RoboDK station: kr30 cnc template half inch flat end mill - paulina 2.rdk

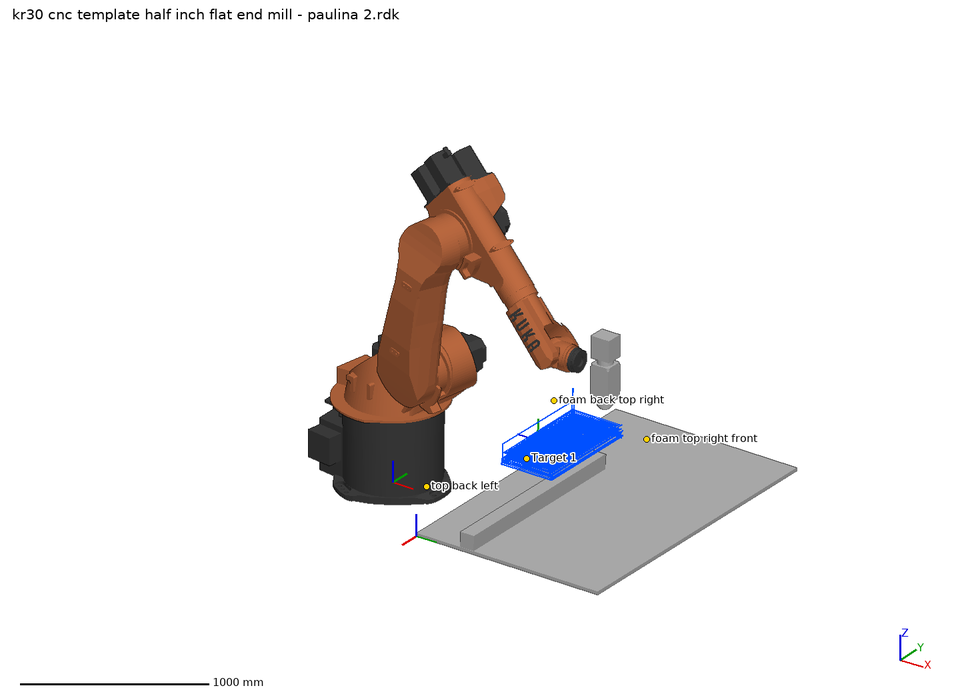
[picture v0: the station drawn from its stored meshes, robots at their saved joint values, targets as dots, program paths as lines]
Station kr30 cnc template half inch flat end mill - paulina 2. Poses are relative to the parent item; angles as X-Y-Z fixed-axis rotations.
  - frame KUKA KR 30 HA Base at (0, 0, 0) mm
    - robot KUKA KR 30 HA: 6 axes, payload 30 kg, reach 2033 mm, repeatability 0.05 mm, weight 665 kg
        modified DH rows (alpha deg, a mm, theta deg, d mm): 0, 0, 0, 815; -90, 350, 0, 0; 0, 850, -90, 0; -90, 145, 0, 820; 90, 0, 0, 0; -90, 0, 180, 170
        joint limits [-185, -135, -120, -350, -119, -350] to [185, 35, 158, 350, 119, 350]; home [0, -90, 90, 0, 0, 0]; saved at [10.988, -78.154, 121.402, 16.012, -43.574, -11.346]
      - tool rc90 spindle mm, TCP at (337.31, -2.2, 160.57) mm, size 110 x 421.3 x 118 mm, geometry from rc90 spindle mm.stl
    - frame Tabletop at (921.82, -1104.91, 385) mm, rotated rx -0.93 ry -0.21 rz -89.9 deg
      - object tabletop CHECK HEIGHT at (-1839.9, 0, 0) mm, size 1839.9 x 1168.4 x 19 mm, geometry from kr30 tabletop mm.stl
      - object kr30 pipe jig base at (-1220, -610.6, 0) mm, size 1217.6 x 88.9 x 88.9 mm, geometry from kr30 pipe jig base.stl
      - frame Frame 3 at (-550, 390, 460) mm, rotated rx 90 ry 0 rz 0 deg
        - target Target 1 (Cartesian target) at (324.46, 69.12, -153.95) mm, rotated rx -179.9 ry 0.14 rz -89.96 deg; joints [37.245, -66.694, 101.534, 53.768, -48.608, -41.204] of KUKA KR 30 HA
    - target foam back top right (Cartesian target) at (1197.65, -230.62, 906.79) mm, rotated rx -15.53 ry 90 rz -15.53 deg; joints [14.757, -102.447, 141.256, 22.791, -41.102, -17.568] of KUKA KR 30 HA
    - target foam top right front (Cartesian target) at (1797.45, -230.62, 850.68) mm, rotated rx -15.58 ry 90 rz -15.58 deg; joints [8.85, -62.405, 99.608, 14.434, -38.093, -11.451] of KUKA KR 30 HA
    - target top back left (Cartesian target) at (1223.08, -1440.01, 894.96) mm, rotated rx 58.97 ry 90 rz 58.97 deg; joints [58.171, -50.232, 76.73, 74.515, -61.834, -59.599] of KUKA KR 30 HA
  - machining project Machining Settings: C:/Users/Research Office/Downloads/B.apt | rotZ(0) | rotX(0)*rotY(0) | roty(-90)
  - program Machining (5196 instructions, listed below)
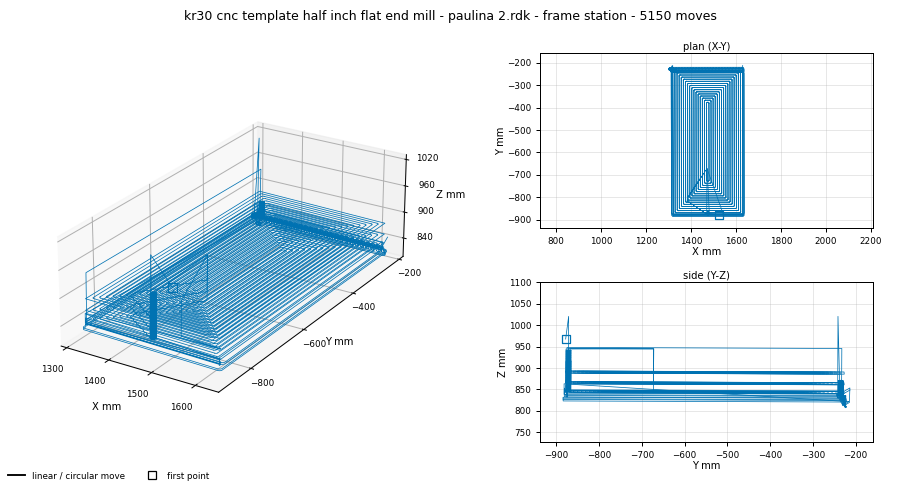
[picture p0: tool path of kr30 cnc template half inch flat end mill - paulina 2.rdk in frame station, 5150 of 5150 moves have a stored position in this frame; points joined in program order, loops and branches not executed]

--- program Machining (robot KUKA KR 30 HA) ---
  Smooth(15)
  Print: /'1001'
  Print: /''
  Print: /'Pocket1'
  Call SetTool(1)
  Set speed (1000.0 mm/s)
  Set Ref.: Frame 3
  Set Tool: rc90 spindle mm
  Show rc90 spindle mm
  MoveJ 1 to (326.02, 133.41, -204.56) mm, rotated rx -179.9 ry 0.15 rz -89.95 deg; joints [36.075, -65.683, 95.357, 56.596, -44.843, -46.24]
  MoveL 2 to (319.15, 185.52, -150.09) mm, rotated rx -179.9 ry 0 rz -90 deg; joints [37.098, -69.807, 97.257, -120.358, 44.337, 130.231]
  MoveL 3 to (319.15, 185.52, -150.09) mm, rotated rx -179.9 ry 0 rz -90 deg; joints [37.098, -69.807, 97.257, -120.358, 44.337, 130.231]
  Set speed (1000.0 mm/s)
  MoveL 4 to (319.15, 108.04, -150.09) mm, rotated rx -179.9 ry 0 rz -90 deg; joints [37.137, -68.08, 100.527, -124.443, 47.047, 136.103]
  Set speed (100.0 mm/s)
  MoveL 5 to (319.13, 107.83, -150.09) mm, rotated rx -179.9 ry 0 rz -90 deg; joints [37.137, -68.075, 100.537, -124.454, 47.054, 136.119]
  MoveL 6 to (319.08, 107.62, -150.09) mm, rotated rx -179.9 ry 0 rz -90 deg; joints [37.135, -68.072, 100.548, -124.467, 47.061, 136.136]
  MoveL 7 to (318.99, 107.42, -150.09) mm, rotated rx -179.9 ry 0 rz -90 deg; joints [37.132, -68.071, 100.56, -124.48, 47.067, 136.154]
  MoveL 8 to (318.86, 107.24, -150.09) mm, rotated rx -179.9 ry 0 rz -90 deg; joints [37.129, -68.071, 100.574, -124.494, 47.072, 136.171]
  MoveL 9 to (318.71, 107.09, -150.1) mm, rotated rx -179.9 ry 0 rz -90 deg; joints [37.124, -68.072, 100.587, -124.508, 47.076, 136.188]
  MoveL 10 to (318.54, 106.96, -150.11) mm, rotated rx -179.9 ry 0 rz -90 deg; joints [37.118, -68.075, 100.601, -124.522, 47.078, 136.204]
  MoveL 11 to (318.35, 106.86, -150.13) mm, rotated rx -179.9 ry 0 rz -90 deg; joints [37.111, -68.078, 100.613, -124.535, 47.078, 136.218]
  MoveL 12 to (318.14, 106.8, -150.16) mm, rotated rx -179.9 ry 0 rz -90 deg; joints [37.104, -68.083, 100.625, -124.547, 47.077, 136.23]
  MoveL 13 to (317.93, 106.77, -150.19) mm, rotated rx -179.9 ry 0 rz -90 deg; joints [37.097, -68.089, 100.634, -124.558, 47.074, 136.24]
  MoveL 14 to (315.89, 106.7, -150.99) mm, rotated rx -179.9 ry 0 rz -90 deg; joints [37.013, -68.123, 100.691, -124.657, 47.028, 136.319]
  MoveL 15 to (314.27, 106.62, -152.45) mm, rotated rx -179.9 ry 0 rz -90 deg; joints [36.926, -68.109, 100.678, -124.744, 46.969, 136.378]
  MoveL 16 to (313.28, 106.54, -154.4) mm, rotated rx -179.9 ry 0 rz -90 deg; joints [36.848, -68.046, 100.598, -124.808, 46.905, 136.41]
  MoveL 17 to (313.05, 106.47, -156.57) mm, rotated rx -179.9 ry 0 rz -90 deg; joints [36.788, -67.944, 100.461, -124.84, 46.845, 136.411]
  MoveL 18 to (313.61, 106.39, -158.69) mm, rotated rx -179.9 ry 0 rz -90 deg; joints [36.756, -67.815, 100.287, -124.838, 46.796, 136.381]
  MoveL 19 to (314.88, 106.31, -160.46) mm, rotated rx -179.9 ry 0 rz -90 deg; joints [36.754, -67.676, 100.098, -124.8, 46.766, 136.325]
  MoveL 20 to (316.71, 106.24, -161.67) mm, rotated rx -179.9 ry 0 rz -90 deg; joints [36.783, -67.546, 99.919, -124.734, 46.759, 136.252]
  MoveL 21 to (318.84, 106.16, -162.15) mm, rotated rx -179.9 ry 0 rz -90 deg; joints [36.84, -67.44, 99.775, -124.649, 46.776, 136.171]
  MoveL 22 to (321, 106.08, -161.83) mm, rotated rx -179.9 ry 0 rz -90 deg; joints [36.915, -67.373, 99.684, -124.556, 46.815, 136.094]
  MoveL 23 to (322.91, 106.01, -160.77) mm, rotated rx -179.9 ry 0 rz -90 deg; joints [37.001, -67.353, 99.659, -124.468, 46.872, 136.033]
  MoveL 24 to (324.31, 105.93, -159.1) mm, rotated rx -179.9 ry 0 rz -90 deg; joints [37.085, -67.382, 99.704, -124.397, 46.94, 135.995]
  MoveL 25 to (325.03, 105.85, -157.03) mm, rotated rx -179.9 ry 0 rz -90 deg; joints [37.158, -67.457, 99.813, -124.353, 47.009, 135.987]
  MoveL 26 to (324.97, 105.78, -154.85) mm, rotated rx -179.9 ry 0 rz -90 deg; joints [37.208, -67.566, 99.972, -124.342, 47.072, 136.01]
  MoveL 27 to (324.13, 105.7, -152.83) mm, rotated rx -179.9 ry 0 rz -90 deg; joints [37.23, -67.697, 100.161, -124.365, 47.121, 136.061]
  MoveL 28 to (322.62, 105.62, -151.24) mm, rotated rx -179.9 ry 0 rz -90 deg; joints [37.221, -67.831, 100.355, -124.42, 47.148, 136.135]
  MoveL 29 to (320.65, 105.55, -150.3) mm, rotated rx -179.9 ry 0 rz -90 deg; joints [37.181, -67.95, 100.529, -124.501, 47.152, 136.222]
  MoveL 30 to (318.48, 105.47, -150.11) mm, rotated rx -179.9 ry 0 rz -90 deg; joints [37.117, -68.039, 100.661, -124.597, 47.131, 136.313]
  MoveL 31 to (316.38, 105.39, -150.72) mm, rotated rx -179.9 ry 0 rz -90 deg; joints [37.035, -68.086, 100.734, -124.697, 47.09, 136.396]
  MoveL 32 to (314.63, 105.32, -152.03) mm, rotated rx -179.9 ry 0 rz -90 deg; joints [36.948, -68.084, 100.739, -124.788, 47.034, 136.46]
  MoveL 33 to (313.47, 105.24, -153.88) mm, rotated rx -179.9 ry 0 rz -90 deg; joints [36.867, -68.033, 100.675, -124.859, 46.97, 136.499]
  MoveL 34 to (313.04, 105.16, -156.02) mm, rotated rx -179.9 ry 0 rz -90 deg; joints [36.802, -67.939, 100.551, -124.9, 46.908, 136.508]
  MoveL 35 to (313.4, 105.09, -158.18) mm, rotated rx -179.9 ry 0 rz -90 deg; joints [36.762, -67.816, 100.385, -124.906, 46.856, 136.486]
  MoveL 36 to (314.5, 105.01, -160.06) mm, rotated rx -179.9 ry 0 rz -90 deg; joints [36.752, -67.678, 100.197, -124.877, 46.82, 136.436]
  MoveL 37 to (316.21, 104.93, -161.43) mm, rotated rx -179.9 ry 0 rz -90 deg; joints [36.774, -67.544, 100.013, -124.818, 46.807, 136.366]
  MoveL 38 to (318.29, 104.86, -162.1) mm, rotated rx -179.9 ry 0 rz -90 deg; joints [36.824, -67.43, 99.858, -124.736, 46.818, 136.286]
  MoveL 39 to (320.47, 104.78, -161.99) mm, rotated rx -179.9 ry 0 rz -90 deg; joints [36.896, -67.353, 99.752, -124.644, 46.852, 136.207]
  MoveL 40 to (322.47, 104.7, -161.1) mm, rotated rx -179.9 ry 0 rz -90 deg; joints [36.98, -67.32, 99.71, -124.553, 46.905, 136.141]
  MoveL 41 to (324.02, 104.63, -159.56) mm, rotated rx -179.9 ry 0 rz -90 deg; joints [37.066, -67.337, 99.738, -124.477, 46.97, 136.097]
  MoveL 42 to (324.92, 104.55, -157.57) mm, rotated rx -179.9 ry 0 rz -90 deg; joints [37.142, -67.401, 99.832, -124.426, 47.04, 136.081]
  MoveL 43 to (325.06, 104.47, -155.39) mm, rotated rx -179.9 ry 0 rz -90 deg; joints [37.198, -67.503, 99.98, -124.406, 47.106, 136.096]
  MoveL 44 to (324.41, 104.4, -153.31) mm, rotated rx -179.9 ry 0 rz -90 deg; joints [37.228, -67.63, 100.163, -124.42, 47.159, 136.141]
  MoveL 45 to (323.06, 104.32, -151.59) mm, rotated rx -179.9 ry 0 rz -90 deg; joints [37.227, -67.764, 100.359, -124.467, 47.192, 136.21]
  MoveL 46 to (321.18, 104.24, -150.47) mm, rotated rx -179.9 ry 0 rz -90 deg; joints [37.195, -67.889, 100.54, -124.542, 47.202, 136.295]
  MoveL 47 to (319.03, 104.17, -150.09) mm, rotated rx -179.9 ry 0 rz -90 deg; joints [37.136, -67.987, 100.685, -124.636, 47.187, 136.385]
  MoveL 48 to (316.88, 104.09, -150.49) mm, rotated rx -179.9 ry 0 rz -90 deg; joints [37.058, -68.045, 100.774, -124.736, 47.151, 136.471]
  MoveL 49 to (315.02, 104.01, -151.64) mm, rotated rx -179.9 ry 0 rz -90 deg; joints [36.971, -68.055, 100.796, -124.831, 47.098, 136.541]
  MoveL 50 to (313.7, 103.94, -153.37) mm, rotated rx -179.9 ry 0 rz -90 deg; joints [36.887, -68.016, 100.749, -124.908, 47.035, 136.587]
  MoveL 51 to (313.07, 103.86, -155.47) mm, rotated rx -179.9 ry 0 rz -90 deg; joints [36.817, -67.933, 100.639, -124.957, 46.972, 136.604]
  MoveL 52 to (313.23, 103.78, -157.65) mm, rotated rx -179.9 ry 0 rz -90 deg; joints [36.77, -67.815, 100.481, -124.972, 46.916, 136.589]
  MoveL 53 to (314.16, 103.71, -159.63) mm, rotated rx -179.9 ry 0 rz -90 deg; joints [36.752, -67.68, 100.296, -124.952, 46.876, 136.546]
  MoveL 54 to (315.73, 103.63, -161.14) mm, rotated rx -179.9 ry 0 rz -90 deg; joints [36.766, -67.543, 100.109, -124.9, 46.857, 136.48]
  MoveL 55 to (317.74, 103.55, -162) mm, rotated rx -179.9 ry 0 rz -90 deg; joints [36.809, -67.423, 99.945, -124.823, 46.861, 136.401]
  MoveL 56 to (319.92, 103.48, -162.09) mm, rotated rx -179.9 ry 0 rz -90 deg; joints [36.877, -67.335, 99.825, -124.732, 46.889, 136.321]
  MoveL 57 to (322, 103.4, -161.39) mm, rotated rx -179.9 ry 0 rz -90 deg; joints [36.959, -67.291, 99.766, -124.639, 46.938, 136.251]
  MoveL 58 to (323.68, 103.32, -160) mm, rotated rx -179.9 ry 0 rz -90 deg; joints [37.045, -67.295, 99.775, -124.559, 47.001, 136.2]
  MoveL 59 to (324.76, 103.25, -158.11) mm, rotated rx -179.9 ry 0 rz -90 deg; joints [37.125, -67.348, 99.853, -124.5, 47.071, 136.177]
  MoveL 60 to (325.1, 103.17, -155.95) mm, rotated rx -179.9 ry 0 rz -90 deg; joints [37.187, -67.441, 99.989, -124.471, 47.138, 136.184]
  MoveL 61 to (324.64, 103.09, -153.81) mm, rotated rx -179.9 ry 0 rz -90 deg; joints [37.224, -67.563, 100.166, -124.477, 47.195, 136.222]
  MoveL 62 to (323.45, 103.02, -151.98) mm, rotated rx -179.9 ry 0 rz -90 deg; joints [37.231, -67.697, 100.361, -124.517, 47.234, 136.285]
  MoveL 63 to (321.69, 102.94, -150.69) mm, rotated rx -179.9 ry 0 rz -90 deg; joints [37.206, -67.826, 100.548, -124.585, 47.25, 136.367]
  MoveL 64 to (319.58, 102.86, -150.11) mm, rotated rx -179.9 ry 0 rz -90 deg; joints [37.153, -67.932, 100.704, -124.675, 47.242, 136.457]
  MoveL 65 to (317.41, 102.79, -150.32) mm, rotated rx -179.9 ry 0 rz -90 deg; joints [37.079, -68.001, 100.808, -124.775, 47.211, 136.545]
  MoveL 66 to (315.45, 102.71, -151.29) mm, rotated rx -179.9 ry 0 rz -90 deg; joints [36.994, -68.024, 100.848, -124.872, 47.161, 136.62]
  MoveL 67 to (313.97, 102.63, -152.89) mm, rotated rx -179.9 ry 0 rz -90 deg; joints [36.908, -67.997, 100.818, -124.955, 47.1, 136.673]
  MoveL 68 to (313.16, 102.56, -154.92) mm, rotated rx -179.9 ry 0 rz -90 deg; joints [36.833, -67.924, 100.723, -125.012, 47.037, 136.697]
  MoveL 69 to (313.12, 102.48, -157.11) mm, rotated rx -179.9 ry 0 rz -90 deg; joints [36.78, -67.814, 100.575, -125.036, 46.978, 136.69]
  MoveL 70 to (313.86, 102.4, -159.16) mm, rotated rx -179.9 ry 0 rz -90 deg; joints [36.754, -67.681, 100.395, -125.025, 46.933, 136.654]
  MoveL 71 to (315.29, 102.33, -160.82) mm, rotated rx -179.9 ry 0 rz -90 deg; joints [36.76, -67.543, 100.206, -124.98, 46.908, 136.593]
  MoveL 72 to (317.21, 102.25, -161.86) mm, rotated rx -179.9 ry 0 rz -90 deg; joints [36.797, -67.417, 100.034, -124.908, 46.907, 136.516]
  MoveL 73 to (319.37, 102.17, -162.14) mm, rotated rx -179.9 ry 0 rz -90 deg; joints [36.859, -67.32, 99.901, -124.819, 46.929, 136.435]
  MoveL 74 to (321.5, 102.1, -161.64) mm, rotated rx -179.9 ry 0 rz -90 deg; joints [36.938, -67.264, 99.825, -124.726, 46.973, 136.361]
  MoveL 75 to (323.31, 102.02, -160.41) mm, rotated rx -179.9 ry 0 rz -90 deg; joints [37.024, -67.256, 99.818, -124.641, 47.033, 136.305]
  MoveL 76 to (324.56, 101.94, -158.62) mm, rotated rx -179.9 ry 0 rz -90 deg; joints [37.107, -67.297, 99.879, -124.576, 47.102, 136.274]
  MoveL 77 to (325.09, 101.86, -156.5) mm, rotated rx -179.9 ry 0 rz -90 deg; joints [37.174, -67.381, 100.002, -124.539, 47.17, 136.274]
  MoveL 78 to (324.83, 101.79, -154.33) mm, rotated rx -179.9 ry 0 rz -90 deg; joints [37.218, -67.497, 100.17, -124.536, 47.231, 136.304]
  MoveL 79 to (323.82, 101.71, -152.4) mm, rotated rx -179.9 ry 0 rz -90 deg; joints [37.233, -67.63, 100.363, -124.567, 47.275, 136.361]
  MoveL 80 to (322.18, 101.63, -150.95) mm, rotated rx -179.9 ry 0 rz -90 deg; joints [37.216, -67.761, 100.554, -124.629, 47.297, 136.439]
  MoveL 81 to (320.13, 101.56, -150.18) mm, rotated rx -179.9 ry 0 rz -90 deg; joints [37.17, -67.875, 100.72, -124.715, 47.295, 136.528]
  MoveL 82 to (317.95, 101.48, -150.19) mm, rotated rx -179.9 ry 0 rz -90 deg; joints [37.1, -67.954, 100.839, -124.813, 47.269, 136.618]
  MoveL 83 to (315.91, 101.4, -150.98) mm, rotated rx -179.9 ry 0 rz -90 deg; joints [37.016, -67.989, 100.896, -124.912, 47.224, 136.697]
  MoveL 84 to (314.29, 101.33, -152.44) mm, rotated rx -179.9 ry 0 rz -90 deg; joints [36.929, -67.975, 100.883, -125, 47.166, 136.756]
  MoveL 85 to (313.29, 101.25, -154.38) mm, rotated rx -179.9 ry 0 rz -90 deg; joints [36.851, -67.913, 100.804, -125.064, 47.102, 136.788]
  MoveL 86 to (313.05, 101.17, -156.56) mm, rotated rx -179.9 ry 0 rz -90 deg; joints [36.792, -67.811, 100.668, -125.097, 47.041, 136.789]
  MoveL 87 to (313.6, 101.1, -158.67) mm, rotated rx -179.9 ry 0 rz -90 deg; joints [36.759, -67.682, 100.493, -125.095, 46.992, 136.76]
  MoveL 88 to (314.87, 101.02, -160.45) mm, rotated rx -179.9 ry 0 rz -90 deg; joints [36.757, -67.544, 100.304, -125.058, 46.962, 136.704]
  MoveL 89 to (316.69, 100.94, -161.66) mm, rotated rx -179.9 ry 0 rz -90 deg; joints [36.786, -67.414, 100.125, -124.992, 46.954, 136.631]
  MoveL 90 to (318.82, 100.87, -162.14) mm, rotated rx -179.9 ry 0 rz -90 deg; joints [36.842, -67.308, 99.981, -124.907, 46.97, 136.55]
  MoveL 91 to (320.98, 100.79, -161.84) mm, rotated rx -179.9 ry 0 rz -90 deg; joints [36.917, -67.241, 99.889, -124.813, 47.008, 136.473]
  MoveL 92 to (322.89, 100.71, -160.78) mm, rotated rx -179.9 ry 0 rz -90 deg; joints [37.003, -67.22, 99.864, -124.725, 47.065, 136.411]
  MoveL 93 to (324.3, 100.64, -159.11) mm, rotated rx -179.9 ry 0 rz -90 deg; joints [37.087, -67.249, 99.908, -124.654, 47.132, 136.374]
  MoveL 94 to (325.03, 100.56, -157.05) mm, rotated rx -179.9 ry 0 rz -90 deg; joints [37.16, -67.323, 100.017, -124.609, 47.202, 136.365]
  MoveL 95 to (324.97, 100.48, -154.87) mm, rotated rx -179.9 ry 0 rz -90 deg; joints [37.21, -67.432, 100.175, -124.597, 47.265, 136.388]
  MoveL 96 to (324.14, 100.41, -152.85) mm, rotated rx -179.9 ry 0 rz -90 deg; joints [37.233, -67.562, 100.364, -124.62, 47.314, 136.439]
  MoveL 97 to (322.64, 100.33, -151.26) mm, rotated rx -179.9 ry 0 rz -90 deg; joints [37.224, -67.696, 100.558, -124.675, 47.342, 136.513]
  MoveL 98 to (320.67, 100.25, -150.3) mm, rotated rx -179.9 ry 0 rz -90 deg; joints [37.184, -67.815, 100.733, -124.755, 47.346, 136.6]
  MoveL 99 to (318.5, 100.18, -150.11) mm, rotated rx -179.9 ry 0 rz -90 deg; joints [37.12, -67.904, 100.865, -124.851, 47.327, 136.69]
  MoveL 100 to (316.39, 100.1, -150.71) mm, rotated rx -179.9 ry 0 rz -90 deg; joints [37.039, -67.951, 100.939, -124.952, 47.286, 136.773]
  MoveL 101 to (314.64, 100.02, -152.02) mm, rotated rx -179.9 ry 0 rz -90 deg; joints [36.952, -67.949, 100.944, -125.043, 47.23, 136.838]
  MoveL 102 to (313.47, 99.95, -153.86) mm, rotated rx -179.9 ry 0 rz -90 deg; joints [36.87, -67.899, 100.88, -125.114, 47.167, 136.877]
  MoveL 103 to (313.04, 99.87, -156) mm, rotated rx -179.9 ry 0 rz -90 deg; joints [36.805, -67.806, 100.757, -125.156, 47.105, 136.886]
  MoveL 104 to (313.39, 99.79, -158.16) mm, rotated rx -179.9 ry 0 rz -90 deg; joints [36.765, -67.683, 100.591, -125.163, 47.052, 136.864]
  MoveL 105 to (314.49, 99.72, -160.05) mm, rotated rx -179.9 ry 0 rz -90 deg; joints [36.755, -67.545, 100.403, -125.134, 47.016, 136.815]
  MoveL 106 to (316.19, 99.64, -161.42) mm, rotated rx -179.9 ry 0 rz -90 deg; joints [36.776, -67.411, 100.219, -125.075, 47.002, 136.745]
  MoveL 107 to (318.27, 99.56, -162.1) mm, rotated rx -179.9 ry 0 rz -90 deg; joints [36.826, -67.298, 100.064, -124.993, 47.012, 136.664]
  MoveL 108 to (320.45, 99.49, -161.99) mm, rotated rx -179.9 ry 0 rz -90 deg; joints [36.898, -67.22, 99.957, -124.901, 47.045, 136.585]
  MoveL 109 to (322.45, 99.41, -161.11) mm, rotated rx -179.9 ry 0 rz -90 deg; joints [36.982, -67.187, 99.915, -124.81, 47.098, 136.519]
  MoveL 110 to (324.01, 99.33, -159.58) mm, rotated rx -179.9 ry 0 rz -90 deg; joints [37.068, -67.204, 99.941, -124.733, 47.163, 136.475]
  MoveL 111 to (324.92, 99.26, -157.59) mm, rotated rx -179.9 ry 0 rz -90 deg; joints [37.144, -67.267, 100.035, -124.681, 47.233, 136.459]
  MoveL 112 to (325.06, 99.18, -155.41) mm, rotated rx -179.9 ry 0 rz -90 deg; joints [37.201, -67.368, 100.182, -124.661, 47.299, 136.474]
  MoveL 113 to (324.42, 99.1, -153.33) mm, rotated rx -179.9 ry 0 rz -90 deg; joints [37.231, -67.494, 100.366, -124.675, 47.352, 136.518]
  MoveL 114 to (323.07, 99.03, -151.6) mm, rotated rx -179.9 ry 0 rz -90 deg; joints [37.23, -67.629, 100.561, -124.722, 47.386, 136.586]
  MoveL 115 to (321.2, 98.95, -150.47) mm, rotated rx -179.9 ry 0 rz -90 deg; joints [37.198, -67.753, 100.743, -124.796, 47.396, 136.671]
  MoveL 116 to (319.05, 98.87, -150.09) mm, rotated rx -179.9 ry 0 rz -90 deg; joints [37.139, -67.851, 100.888, -124.89, 47.383, 136.762]
  MoveL 117 to (316.9, 98.8, -150.49) mm, rotated rx -179.9 ry 0 rz -90 deg; joints [37.061, -67.91, 100.977, -124.99, 47.347, 136.847]
  MoveL 118 to (315.04, 98.72, -151.63) mm, rotated rx -179.9 ry 0 rz -90 deg; joints [36.974, -67.92, 101, -125.085, 47.295, 136.917]
  MoveL 119 to (313.7, 98.64, -153.36) mm, rotated rx -179.9 ry 0 rz -90 deg; joints [36.89, -67.882, 100.953, -125.162, 47.232, 136.964]
  MoveL 120 to (313.07, 98.57, -155.45) mm, rotated rx -179.9 ry 0 rz -90 deg; joints [36.82, -67.799, 100.844, -125.212, 47.169, 136.981]
  MoveL 121 to (313.23, 98.49, -157.63) mm, rotated rx -179.9 ry 0 rz -90 deg; joints [36.773, -67.682, 100.686, -125.228, 47.113, 136.966]
  MoveL 122 to (314.15, 98.41, -159.61) mm, rotated rx -179.9 ry 0 rz -90 deg; joints [36.755, -67.546, 100.502, -125.208, 47.073, 136.923]
  MoveL 123 to (315.72, 98.34, -161.13) mm, rotated rx -179.9 ry 0 rz -90 deg; joints [36.769, -67.41, 100.314, -125.156, 47.053, 136.858]
  MoveL 124 to (317.72, 98.26, -162) mm, rotated rx -179.9 ry 0 rz -90 deg; joints [36.812, -67.29, 100.15, -125.079, 47.056, 136.779]
  MoveL 125 to (319.91, 98.18, -162.09) mm, rotated rx -179.9 ry 0 rz -90 deg; joints [36.879, -67.202, 100.029, -124.988, 47.084, 136.699]
  MoveL 126 to (321.98, 98.11, -161.4) mm, rotated rx -179.9 ry 0 rz -90 deg; joints [36.961, -67.157, 99.97, -124.896, 47.132, 136.628]
  MoveL 127 to (323.67, 98.03, -160.02) mm, rotated rx -179.9 ry 0 rz -90 deg; joints [37.047, -67.161, 99.979, -124.814, 47.194, 136.577]
  MoveL 128 to (324.76, 97.95, -158.12) mm, rotated rx -179.9 ry 0 rz -90 deg; joints [37.127, -67.213, 100.056, -124.755, 47.264, 136.554]
  MoveL 129 to (325.1, 97.88, -155.97) mm, rotated rx -179.9 ry 0 rz -90 deg; joints [37.189, -67.306, 100.192, -124.726, 47.332, 136.561]
  MoveL 130 to (324.65, 97.8, -153.83) mm, rotated rx -179.9 ry 0 rz -90 deg; joints [37.227, -67.427, 100.368, -124.731, 47.389, 136.598]
  MoveL 131 to (323.47, 97.72, -151.99) mm, rotated rx -179.9 ry 0 rz -90 deg; joints [37.233, -67.561, 100.563, -124.77, 47.428, 136.661]
  MoveL 132 to (321.71, 97.65, -150.69) mm, rotated rx -179.9 ry 0 rz -90 deg; joints [37.209, -67.69, 100.75, -124.838, 47.445, 136.743]
  MoveL 133 to (319.6, 97.57, -150.11) mm, rotated rx -179.9 ry 0 rz -90 deg; joints [37.157, -67.796, 100.906, -124.928, 47.437, 136.833]
  MoveL 134 to (317.43, 97.49, -150.31) mm, rotated rx -179.9 ry 0 rz -90 deg; joints [37.083, -67.865, 101.011, -125.028, 47.407, 136.921]
  MoveL 135 to (315.47, 97.41, -151.28) mm, rotated rx -179.9 ry 0 rz -90 deg; joints [36.997, -67.888, 101.051, -125.125, 47.358, 136.996]
  MoveL 136 to (313.98, 97.34, -152.88) mm, rotated rx -179.9 ry 0 rz -90 deg; joints [36.911, -67.862, 101.022, -125.208, 47.298, 137.049]
  MoveL 137 to (313.16, 97.26, -154.9) mm, rotated rx -179.9 ry 0 rz -90 deg; joints [36.837, -67.789, 100.927, -125.266, 47.234, 137.073]
  MoveL 138 to (313.11, 97.18, -157.09) mm, rotated rx -179.9 ry 0 rz -90 deg; joints [36.783, -67.68, 100.78, -125.291, 47.176, 137.067]
  MoveL 139 to (313.85, 97.11, -159.14) mm, rotated rx -179.9 ry 0 rz -90 deg; joints [36.757, -67.547, 100.6, -125.28, 47.13, 137.03]
  MoveL 140 to (315.27, 97.03, -160.8) mm, rotated rx -179.9 ry 0 rz -90 deg; joints [36.763, -67.409, 100.411, -125.236, 47.105, 136.97]
  MoveL 141 to (317.19, 96.95, -161.85) mm, rotated rx -179.9 ry 0 rz -90 deg; joints [36.799, -67.284, 100.238, -125.164, 47.102, 136.893]
  MoveL 142 to (319.35, 96.88, -162.14) mm, rotated rx -179.9 ry 0 rz -90 deg; joints [36.861, -67.187, 100.105, -125.075, 47.124, 136.812]
  MoveL 143 to (321.48, 96.8, -161.65) mm, rotated rx -179.9 ry 0 rz -90 deg; joints [36.94, -67.13, 100.029, -124.982, 47.167, 136.738]
  MoveL 144 to (323.29, 96.72, -160.42) mm, rotated rx -179.9 ry 0 rz -90 deg; joints [37.026, -67.122, 100.02, -124.897, 47.226, 136.682]
  MoveL 145 to (324.55, 96.65, -158.64) mm, rotated rx -179.9 ry 0 rz -90 deg; joints [37.109, -67.162, 100.081, -124.831, 47.295, 136.651]
  MoveL 146 to (325.09, 96.57, -156.52) mm, rotated rx -179.9 ry 0 rz -90 deg; joints [37.176, -67.245, 100.203, -124.793, 47.364, 136.65]
  MoveL 147 to (324.84, 96.49, -154.35) mm, rotated rx -179.9 ry 0 rz -90 deg; joints [37.221, -67.361, 100.372, -124.79, 47.424, 136.68]
  MoveL 148 to (323.83, 96.42, -152.41) mm, rotated rx -179.9 ry 0 rz -90 deg; joints [37.235, -67.493, 100.564, -124.82, 47.469, 136.737]
  MoveL 149 to (322.19, 96.34, -150.96) mm, rotated rx -179.9 ry 0 rz -90 deg; joints [37.219, -67.625, 100.755, -124.882, 47.492, 136.815]
  MoveL 150 to (320.15, 96.26, -150.18) mm, rotated rx -179.9 ry 0 rz -90 deg; joints [37.173, -67.738, 100.922, -124.967, 47.49, 136.904]
  MoveL 151 to (317.97, 96.19, -150.19) mm, rotated rx -179.9 ry 0 rz -90 deg; joints [37.103, -67.818, 101.041, -125.065, 47.466, 136.993]
  MoveL 152 to (315.93, 96.11, -150.97) mm, rotated rx -179.9 ry 0 rz -90 deg; joints [37.02, -67.853, 101.098, -125.165, 47.421, 137.072]
  MoveL 153 to (314.3, 96.03, -152.42) mm, rotated rx -179.9 ry 0 rz -90 deg; joints [36.933, -67.839, 101.086, -125.252, 47.363, 137.131]
  MoveL 154 to (313.3, 95.96, -154.37) mm, rotated rx -179.9 ry 0 rz -90 deg; joints [36.854, -67.777, 101.007, -125.317, 47.299, 137.164]
  MoveL 155 to (313.05, 95.88, -156.54) mm, rotated rx -179.9 ry 0 rz -90 deg; joints [36.795, -67.676, 100.872, -125.351, 47.239, 137.165]
  MoveL 156 to (313.59, 95.8, -158.65) mm, rotated rx -179.9 ry 0 rz -90 deg; joints [36.761, -67.548, 100.698, -125.349, 47.189, 137.136]
  MoveL 157 to (314.86, 95.73, -160.44) mm, rotated rx -179.9 ry 0 rz -90 deg; joints [36.759, -67.41, 100.509, -125.313, 47.158, 137.08]
  MoveL 158 to (316.67, 95.65, -161.65) mm, rotated rx -179.9 ry 0 rz -90 deg; joints [36.788, -67.28, 100.329, -125.247, 47.15, 137.007]
  MoveL 159 to (318.8, 95.57, -162.14) mm, rotated rx -179.9 ry 0 rz -90 deg; joints [36.844, -67.174, 100.184, -125.162, 47.165, 136.926]
  MoveL 160 to (320.96, 95.5, -161.84) mm, rotated rx -179.9 ry 0 rz -90 deg; joints [36.919, -67.106, 100.092, -125.068, 47.203, 136.849]
  MoveL 161 to (322.88, 95.42, -160.79) mm, rotated rx -179.9 ry 0 rz -90 deg; joints [37.005, -67.085, 100.066, -124.98, 47.259, 136.787]
  MoveL 162 to (324.3, 95.34, -159.13) mm, rotated rx -179.9 ry 0 rz -90 deg; joints [37.089, -67.114, 100.11, -124.908, 47.326, 136.749]
  MoveL 163 to (325.03, 95.27, -157.07) mm, rotated rx -179.9 ry 0 rz -90 deg; joints [37.162, -67.187, 100.218, -124.863, 47.395, 136.741]
  MoveL 164 to (324.97, 95.19, -154.89) mm, rotated rx -179.9 ry 0 rz -90 deg; joints [37.213, -67.296, 100.376, -124.85, 47.459, 136.763]
  MoveL 165 to (324.15, 95.11, -152.86) mm, rotated rx -179.9 ry 0 rz -90 deg; joints [37.235, -67.425, 100.565, -124.872, 47.508, 136.814]
  MoveL 166 to (322.65, 95.04, -151.27) mm, rotated rx -179.9 ry 0 rz -90 deg; joints [37.227, -67.559, 100.759, -124.927, 47.537, 136.887]
  MoveL 167 to (320.69, 94.96, -150.31) mm, rotated rx -179.9 ry 0 rz -90 deg; joints [37.188, -67.678, 100.934, -125.007, 47.542, 136.974]
  MoveL 168 to (318.52, 94.88, -150.11) mm, rotated rx -179.9 ry 0 rz -90 deg; joints [37.123, -67.767, 101.067, -125.103, 47.523, 137.065]
  MoveL 169 to (316.41, 94.81, -150.7) mm, rotated rx -179.9 ry 0 rz -90 deg; joints [37.042, -67.814, 101.141, -125.203, 47.483, 137.147]
  MoveL 170 to (314.66, 94.73, -152) mm, rotated rx -179.9 ry 0 rz -90 deg; joints [36.955, -67.813, 101.146, -125.295, 47.428, 137.212]
  MoveL 171 to (313.48, 94.65, -153.84) mm, rotated rx -179.9 ry 0 rz -90 deg; joints [36.873, -67.763, 101.083, -125.367, 47.365, 137.252]
  MoveL 172 to (313.04, 94.58, -155.98) mm, rotated rx -179.9 ry 0 rz -90 deg; joints [36.808, -67.67, 100.961, -125.409, 47.303, 137.261]
  MoveL 173 to (313.38, 94.5, -158.14) mm, rotated rx -179.9 ry 0 rz -90 deg; joints [36.768, -67.548, 100.794, -125.416, 47.25, 137.239]
  MoveL 174 to (314.48, 94.42, -160.03) mm, rotated rx -179.9 ry 0 rz -90 deg; joints [36.757, -67.41, 100.607, -125.388, 47.214, 137.19]
  MoveL 175 to (316.17, 94.35, -161.41) mm, rotated rx -179.9 ry 0 rz -90 deg; joints [36.779, -67.277, 100.423, -125.329, 47.199, 137.12]
  MoveL 176 to (318.25, 94.27, -162.09) mm, rotated rx -179.9 ry 0 rz -90 deg; joints [36.828, -67.163, 100.267, -125.248, 47.208, 137.04]
  MoveL 177 to (320.43, 94.19, -161.99) mm, rotated rx -179.9 ry 0 rz -90 deg; joints [36.9, -67.085, 100.16, -125.155, 47.24, 136.961]
  MoveL 178 to (322.43, 94.12, -161.12) mm, rotated rx -179.9 ry 0 rz -90 deg; joints [36.984, -67.052, 100.117, -125.064, 47.292, 136.894]
  MoveL 179 to (324, 94.04, -159.6) mm, rotated rx -179.9 ry 0 rz -90 deg; joints [37.069, -67.068, 100.143, -124.987, 47.357, 136.85]
  MoveL 180 to (324.91, 93.96, -157.61) mm, rotated rx -179.9 ry 0 rz -90 deg; joints [37.146, -67.131, 100.235, -124.934, 47.427, 136.834]
  MoveL 181 to (325.06, 93.89, -155.43) mm, rotated rx -179.9 ry 0 rz -90 deg; joints [37.203, -67.232, 100.383, -124.913, 47.493, 136.848]
  MoveL 182 to (324.42, 93.81, -153.34) mm, rotated rx -179.9 ry 0 rz -90 deg; joints [37.233, -67.357, 100.566, -124.926, 47.546, 136.892]
  MoveL 183 to (323.08, 93.73, -151.62) mm, rotated rx -179.9 ry 0 rz -90 deg; joints [37.232, -67.491, 100.761, -124.973, 47.581, 136.961]
  MoveL 184 to (321.22, 93.66, -150.48) mm, rotated rx -179.9 ry 0 rz -90 deg; joints [37.201, -67.616, 100.943, -125.047, 47.592, 137.045]
  MoveL 185 to (319.07, 93.58, -150.09) mm, rotated rx -179.9 ry 0 rz -90 deg; joints [37.142, -67.714, 101.088, -125.14, 47.579, 137.136]
  MoveL 186 to (316.92, 93.5, -150.48) mm, rotated rx -179.9 ry 0 rz -90 deg; joints [37.064, -67.772, 101.178, -125.241, 47.544, 137.221]
  MoveL 187 to (315.05, 93.43, -151.62) mm, rotated rx -179.9 ry 0 rz -90 deg; joints [36.978, -67.783, 101.202, -125.336, 47.492, 137.291]
  MoveL 188 to (313.71, 93.35, -153.34) mm, rotated rx -179.9 ry 0 rz -90 deg; joints [36.894, -67.745, 101.156, -125.414, 47.43, 137.338]
  MoveL 189 to (313.07, 93.27, -155.43) mm, rotated rx -179.9 ry 0 rz -90 deg; joints [36.823, -67.662, 101.047, -125.464, 47.367, 137.355]
  MoveL 190 to (313.22, 93.2, -157.61) mm, rotated rx -179.9 ry 0 rz -90 deg; joints [36.776, -67.546, 100.889, -125.481, 47.311, 137.341]
  MoveL 191 to (314.14, 93.12, -159.59) mm, rotated rx -179.9 ry 0 rz -90 deg; joints [36.758, -67.411, 100.705, -125.461, 47.27, 137.298]
  MoveL 192 to (315.7, 93.04, -161.12) mm, rotated rx -179.9 ry 0 rz -90 deg; joints [36.771, -67.275, 100.517, -125.41, 47.25, 137.232]
  MoveL 193 to (317.7, 92.97, -161.99) mm, rotated rx -179.9 ry 0 rz -90 deg; joints [36.814, -67.155, 100.352, -125.333, 47.253, 137.154]
  MoveL 194 to (319.89, 92.89, -162.09) mm, rotated rx -179.9 ry 0 rz -90 deg; joints [36.881, -67.067, 100.231, -125.242, 47.279, 137.074]
  MoveL 195 to (321.96, 92.81, -161.41) mm, rotated rx -179.9 ry 0 rz -90 deg; joints [36.963, -67.022, 100.171, -125.149, 47.327, 137.003]
  MoveL 196 to (323.66, 92.73, -160.03) mm, rotated rx -179.9 ry 0 rz -90 deg; joints [37.049, -67.025, 100.18, -125.067, 47.389, 136.952]
  MoveL 197 to (324.75, 92.66, -158.14) mm, rotated rx -179.9 ry 0 rz -90 deg; joints [37.129, -67.077, 100.256, -125.008, 47.458, 136.928]
  MoveL 198 to (325.1, 92.58, -155.98) mm, rotated rx -179.9 ry 0 rz -90 deg; joints [37.192, -67.169, 100.392, -124.978, 47.526, 136.935]
  MoveL 199 to (324.66, 92.5, -153.84) mm, rotated rx -179.9 ry 0 rz -90 deg; joints [37.229, -67.29, 100.568, -124.982, 47.583, 136.972]
  MoveL 200 to (323.48, 92.43, -152) mm, rotated rx -179.9 ry 0 rz -90 deg; joints [37.236, -67.423, 100.762, -125.021, 47.623, 137.035]
  MoveL 201 to (321.73, 92.35, -150.7) mm, rotated rx -179.9 ry 0 rz -90 deg; joints [37.212, -67.552, 100.95, -125.089, 47.64, 137.116]
  MoveL 202 to (319.62, 92.27, -150.11) mm, rotated rx -179.9 ry 0 rz -90 deg; joints [37.16, -67.658, 101.106, -125.178, 47.634, 137.206]
  MoveL 203 to (317.45, 92.2, -150.31) mm, rotated rx -179.9 ry 0 rz -90 deg; joints [37.086, -67.727, 101.212, -125.278, 47.604, 137.294]
  MoveL 204 to (315.48, 92.12, -151.27) mm, rotated rx -179.9 ry 0 rz -90 deg; joints [37, -67.751, 101.252, -125.376, 47.556, 137.369]
  MoveL 205 to (313.99, 92.04, -152.86) mm, rotated rx -179.9 ry 0 rz -90 deg; joints [36.915, -67.725, 101.224, -125.459, 47.496, 137.422]
  MoveL 206 to (313.16, 91.97, -154.88) mm, rotated rx -179.9 ry 0 rz -90 deg; joints [36.84, -67.652, 101.129, -125.517, 47.432, 137.447]
  MoveL 207 to (313.11, 91.89, -157.07) mm, rotated rx -179.9 ry 0 rz -90 deg; joints [36.786, -67.543, 100.983, -125.543, 47.374, 137.44]
  MoveL 208 to (313.84, 91.81, -159.13) mm, rotated rx -179.9 ry 0 rz -90 deg; joints [36.76, -67.412, 100.803, -125.532, 47.328, 137.404]
  MoveL 209 to (315.26, 91.74, -160.79) mm, rotated rx -179.9 ry 0 rz -90 deg; joints [36.765, -67.274, 100.614, -125.488, 47.302, 137.344]
  MoveL 210 to (317.17, 91.66, -161.84) mm, rotated rx -179.9 ry 0 rz -90 deg; joints [36.801, -67.148, 100.441, -125.417, 47.299, 137.267]
  MoveL 211 to (319.33, 91.58, -162.14) mm, rotated rx -179.9 ry 0 rz -90 deg; joints [36.863, -67.051, 100.307, -125.328, 47.32, 137.186]
  MoveL 212 to (321.46, 91.51, -161.65) mm, rotated rx -179.9 ry 0 rz -90 deg; joints [36.942, -66.994, 100.23, -125.235, 47.362, 137.112]
  MoveL 213 to (323.28, 91.43, -160.44) mm, rotated rx -179.9 ry 0 rz -90 deg; joints [37.028, -66.986, 100.221, -125.149, 47.421, 137.056]
  MoveL 214 to (324.54, 91.35, -158.65) mm, rotated rx -179.9 ry 0 rz -90 deg; joints [37.111, -67.025, 100.281, -125.083, 47.489, 137.024]
  MoveL 215 to (325.09, 91.28, -156.54) mm, rotated rx -179.9 ry 0 rz -90 deg; joints [37.178, -67.108, 100.403, -125.045, 47.558, 137.023]
  MoveL 216 to (324.84, 91.2, -154.37) mm, rotated rx -179.9 ry 0 rz -90 deg; joints [37.223, -67.223, 100.571, -125.04, 47.619, 137.053]
  MoveL 217 to (323.84, 91.12, -152.43) mm, rotated rx -179.9 ry 0 rz -90 deg; joints [37.238, -67.355, 100.763, -125.07, 47.664, 137.11]
  MoveL 218 to (322.21, 91.05, -150.97) mm, rotated rx -179.9 ry 0 rz -90 deg; joints [37.222, -67.486, 100.955, -125.131, 47.687, 137.187]
  MoveL 219 to (320.17, 90.97, -150.19) mm, rotated rx -179.9 ry 0 rz -90 deg; joints [37.176, -67.599, 101.121, -125.216, 47.687, 137.276]
  MoveL 220 to (317.99, 90.89, -150.18) mm, rotated rx -179.9 ry 0 rz -90 deg; joints [37.107, -67.679, 101.241, -125.315, 47.663, 137.366]
  MoveL 221 to (315.94, 90.82, -150.96) mm, rotated rx -179.9 ry 0 rz -90 deg; joints [37.023, -67.715, 101.299, -125.414, 47.619, 137.445]
  MoveL 222 to (314.31, 90.74, -152.41) mm, rotated rx -179.9 ry 0 rz -90 deg; joints [36.936, -67.701, 101.287, -125.503, 47.561, 137.504]
  MoveL 223 to (313.3, 90.66, -154.35) mm, rotated rx -179.9 ry 0 rz -90 deg; joints [36.858, -67.64, 101.209, -125.568, 47.498, 137.536]
  MoveL 224 to (313.05, 90.59, -156.52) mm, rotated rx -179.9 ry 0 rz -90 deg; joints [36.798, -67.539, 101.074, -125.602, 47.437, 137.538]
  MoveL 225 to (313.59, 90.51, -158.64) mm, rotated rx -179.9 ry 0 rz -90 deg; joints [36.764, -67.411, 100.9, -125.601, 47.388, 137.509]
  MoveL 226 to (314.84, 90.43, -160.42) mm, rotated rx -179.9 ry 0 rz -90 deg; joints [36.762, -67.274, 100.711, -125.565, 47.356, 137.454]
  MoveL 227 to (316.65, 90.36, -161.65) mm, rotated rx -179.9 ry 0 rz -90 deg; joints [36.79, -67.144, 100.531, -125.5, 47.347, 137.381]
  MoveL 228 to (318.78, 90.28, -162.14) mm, rotated rx -179.9 ry 0 rz -90 deg; joints [36.846, -67.038, 100.386, -125.414, 47.361, 137.3]
  MoveL 229 to (320.95, 90.2, -161.85) mm, rotated rx -179.9 ry 0 rz -90 deg; joints [36.921, -66.97, 100.293, -125.321, 47.399, 137.223]
  MoveL 230 to (322.87, 90.13, -160.81) mm, rotated rx -179.9 ry 0 rz -90 deg; joints [37.007, -66.949, 100.266, -125.232, 47.454, 137.161]
  MoveL 231 to (324.29, 90.05, -159.15) mm, rotated rx -179.9 ry 0 rz -90 deg; joints [37.091, -66.976, 100.309, -125.159, 47.52, 137.123]
  MoveL 232 to (325.02, 89.97, -157.09) mm, rotated rx -179.9 ry 0 rz -90 deg; joints [37.164, -67.049, 100.417, -125.114, 47.59, 137.114]
  MoveL 233 to (324.98, 89.9, -154.9) mm, rotated rx -179.9 ry 0 rz -90 deg; joints [37.215, -67.157, 100.575, -125.1, 47.654, 137.136]
  MoveL 234 to (324.16, 89.82, -152.88) mm, rotated rx -179.9 ry 0 rz -90 deg; joints [37.238, -67.287, 100.763, -125.122, 47.703, 137.186]
  MoveL 235 to (322.67, 89.74, -151.28) mm, rotated rx -179.9 ry 0 rz -90 deg; joints [37.229, -67.42, 100.957, -125.176, 47.733, 137.259]
  MoveL 236 to (320.71, 89.67, -150.31) mm, rotated rx -179.9 ry 0 rz -90 deg; joints [37.191, -67.539, 101.132, -125.255, 47.739, 137.346]
  MoveL 237 to (318.53, 89.59, -150.11) mm, rotated rx -179.9 ry 0 rz -90 deg; joints [37.127, -67.628, 101.266, -125.352, 47.72, 137.436]
  MoveL 238 to (316.43, 89.51, -150.69) mm, rotated rx -179.9 ry 0 rz -90 deg; joints [37.046, -67.675, 101.34, -125.452, 47.681, 137.519]
  MoveL 239 to (314.67, 89.44, -151.99) mm, rotated rx -179.9 ry 0 rz -90 deg; joints [36.959, -67.674, 101.347, -125.544, 47.626, 137.584]
  MoveL 240 to (313.49, 89.36, -153.83) mm, rotated rx -179.9 ry 0 rz -90 deg; joints [36.877, -67.625, 101.284, -125.616, 47.564, 137.624]
  MoveL 241 to (313.04, 89.28, -155.96) mm, rotated rx -179.9 ry 0 rz -90 deg; joints [36.811, -67.533, 101.162, -125.659, 47.502, 137.633]
  MoveL 242 to (313.38, 89.21, -158.12) mm, rotated rx -179.9 ry 0 rz -90 deg; joints [36.771, -67.411, 100.996, -125.667, 47.449, 137.612]
  MoveL 243 to (314.47, 89.13, -160.02) mm, rotated rx -179.9 ry 0 rz -90 deg; joints [36.76, -67.274, 100.808, -125.64, 47.412, 137.563]
  MoveL 244 to (316.16, 89.05, -161.4) mm, rotated rx -179.9 ry 0 rz -90 deg; joints [36.781, -67.14, 100.624, -125.581, 47.396, 137.493]
  MoveL 245 to (318.23, 88.98, -162.09) mm, rotated rx -179.9 ry 0 rz -90 deg; joints [36.83, -67.027, 100.468, -125.5, 47.405, 137.413]
  MoveL 246 to (320.41, 88.9, -162) mm, rotated rx -179.9 ry 0 rz -90 deg; joints [36.902, -66.949, 100.36, -125.407, 47.436, 137.334]
  MoveL 247 to (322.42, 88.82, -161.13) mm, rotated rx -179.9 ry 0 rz -90 deg; joints [36.986, -66.915, 100.316, -125.315, 47.488, 137.267]
  MoveL 248 to (323.99, 88.75, -159.61) mm, rotated rx -179.9 ry 0 rz -90 deg; joints [37.071, -66.93, 100.342, -125.238, 47.552, 137.222]
  MoveL 249 to (324.91, 88.67, -157.63) mm, rotated rx -179.9 ry 0 rz -90 deg; joints [37.148, -66.993, 100.434, -125.185, 47.622, 137.206]
  MoveL 250 to (325.06, 88.59, -155.45) mm, rotated rx -179.9 ry 0 rz -90 deg; joints [37.205, -67.093, 100.581, -125.163, 47.687, 137.22]
  MoveL 251 to (324.43, 88.52, -153.36) mm, rotated rx -179.9 ry 0 rz -90 deg; joints [37.236, -67.218, 100.764, -125.175, 47.741, 137.264]
  MoveL 252 to (323.1, 88.44, -151.63) mm, rotated rx -179.9 ry 0 rz -90 deg; joints [37.235, -67.352, 100.959, -125.221, 47.777, 137.332]
  MoveL 253 to (321.24, 88.36, -150.49) mm, rotated rx -179.9 ry 0 rz -90 deg; joints [37.204, -67.476, 101.141, -125.295, 47.789, 137.416]
  MoveL 254 to (319.09, 88.29, -150.09) mm, rotated rx -179.9 ry 0 rz -90 deg; joints [37.145, -67.574, 101.287, -125.388, 47.777, 137.507]
  MoveL 255 to (316.94, 88.21, -150.47) mm, rotated rx -179.9 ry 0 rz -90 deg; joints [37.068, -67.633, 101.377, -125.489, 47.742, 137.592]
  MoveL 256 to (315.07, 88.13, -151.6) mm, rotated rx -179.9 ry 0 rz -90 deg; joints [36.981, -67.644, 101.401, -125.585, 47.691, 137.663]
  MoveL 257 to (313.72, 88.05, -153.32) mm, rotated rx -179.9 ry 0 rz -90 deg; joints [36.897, -67.606, 101.356, -125.663, 47.63, 137.709]
  MoveL 258 to (313.08, 87.98, -155.41) mm, rotated rx -179.9 ry 0 rz -90 deg; joints [36.826, -67.524, 101.247, -125.714, 47.567, 137.727]
  MoveL 259 to (313.22, 87.9, -157.59) mm, rotated rx -179.9 ry 0 rz -90 deg; joints [36.779, -67.409, 101.09, -125.731, 47.51, 137.713]
  MoveL 260 to (314.13, 87.82, -159.58) mm, rotated rx -179.9 ry 0 rz -90 deg; joints [36.76, -67.274, 100.906, -125.712, 47.469, 137.67]
  MoveL 261 to (315.68, 87.75, -161.11) mm, rotated rx -179.9 ry 0 rz -90 deg; joints [36.773, -67.138, 100.718, -125.661, 47.448, 137.605]
  MoveL 262 to (317.69, 87.67, -161.99) mm, rotated rx -179.9 ry 0 rz -90 deg; joints [36.816, -67.018, 100.553, -125.584, 47.45, 137.526]
  MoveL 263 to (319.87, 87.59, -162.1) mm, rotated rx -179.9 ry 0 rz -90 deg; joints [36.883, -66.93, 100.431, -125.493, 47.476, 137.446]
  MoveL 264 to (321.95, 87.52, -161.42) mm, rotated rx -179.9 ry 0 rz -90 deg; joints [36.964, -66.884, 100.371, -125.4, 47.522, 137.375]
  MoveL 265 to (323.64, 87.44, -160.05) mm, rotated rx -179.9 ry 0 rz -90 deg; joints [37.051, -66.887, 100.378, -125.318, 47.584, 137.324]
  MoveL 266 to (324.74, 87.36, -158.16) mm, rotated rx -179.9 ry 0 rz -90 deg; joints [37.131, -66.938, 100.455, -125.257, 47.653, 137.3]
  MoveL 267 to (325.1, 87.29, -156) mm, rotated rx -179.9 ry 0 rz -90 deg; joints [37.194, -67.03, 100.589, -125.227, 47.721, 137.306]
  MoveL 268 to (324.66, 87.21, -153.86) mm, rotated rx -179.9 ry 0 rz -90 deg; joints [37.231, -67.15, 100.765, -125.231, 47.778, 137.343]
  MoveL 269 to (323.49, 87.13, -152.02) mm, rotated rx -179.9 ry 0 rz -90 deg; joints [37.239, -67.284, 100.96, -125.269, 47.819, 137.406]
  MoveL 270 to (321.74, 87.06, -150.71) mm, rotated rx -179.9 ry 0 rz -90 deg; joints [37.215, -67.412, 101.147, -125.336, 47.837, 137.487]
  MoveL 271 to (319.64, 86.98, -150.11) mm, rotated rx -179.9 ry 0 rz -90 deg; joints [37.163, -67.518, 101.304, -125.426, 47.831, 137.577]
  MoveL 272 to (317.46, 86.9, -150.3) mm, rotated rx -179.9 ry 0 rz -90 deg; joints [37.089, -67.587, 101.41, -125.526, 47.802, 137.664]
  MoveL 273 to (315.5, 86.83, -151.25) mm, rotated rx -179.9 ry 0 rz -90 deg; joints [37.004, -67.611, 101.451, -125.624, 47.755, 137.739]
  MoveL 274 to (314, 86.75, -152.85) mm, rotated rx -179.9 ry 0 rz -90 deg; joints [36.918, -67.585, 101.423, -125.707, 47.695, 137.793]
  MoveL 275 to (313.17, 86.67, -154.87) mm, rotated rx -179.9 ry 0 rz -90 deg; joints [36.843, -67.514, 101.329, -125.766, 47.632, 137.818]
  MoveL 276 to (313.11, 86.6, -157.05) mm, rotated rx -179.9 ry 0 rz -90 deg; joints [36.789, -67.405, 101.183, -125.792, 47.573, 137.811]
  MoveL 277 to (313.83, 86.52, -159.11) mm, rotated rx -179.9 ry 0 rz -90 deg; joints [36.763, -67.274, 101.003, -125.782, 47.527, 137.776]
  MoveL 278 to (315.24, 86.44, -160.78) mm, rotated rx -179.9 ry 0 rz -90 deg; joints [36.768, -67.136, 100.814, -125.738, 47.5, 137.715]
  MoveL 279 to (317.15, 86.37, -161.84) mm, rotated rx -179.9 ry 0 rz -90 deg; joints [36.803, -67.011, 100.641, -125.667, 47.497, 137.639]
  MoveL 280 to (319.32, 86.29, -162.15) mm, rotated rx -179.9 ry 0 rz -90 deg; joints [36.865, -66.914, 100.506, -125.579, 47.516, 137.558]
  MoveL 281 to (321.45, 86.21, -161.66) mm, rotated rx -179.9 ry 0 rz -90 deg; joints [36.944, -66.857, 100.429, -125.485, 47.558, 137.484]
  MoveL 282 to (323.27, 86.14, -160.45) mm, rotated rx -179.9 ry 0 rz -90 deg; joints [37.03, -66.847, 100.419, -125.399, 47.617, 137.427]
  MoveL 283 to (324.53, 86.06, -158.67) mm, rotated rx -179.9 ry 0 rz -90 deg; joints [37.113, -66.886, 100.479, -125.332, 47.685, 137.395]
  MoveL 284 to (325.08, 85.98, -156.56) mm, rotated rx -179.9 ry 0 rz -90 deg; joints [37.181, -66.969, 100.6, -125.293, 47.753, 137.394]
  MoveL 285 to (324.85, 85.91, -154.39) mm, rotated rx -179.9 ry 0 rz -90 deg; joints [37.225, -67.083, 100.768, -125.288, 47.814, 137.423]
  MoveL 286 to (323.85, 85.83, -152.44) mm, rotated rx -179.9 ry 0 rz -90 deg; joints [37.241, -67.215, 100.96, -125.318, 47.86, 137.48]
  MoveL 287 to (322.23, 85.75, -150.98) mm, rotated rx -179.9 ry 0 rz -90 deg; joints [37.225, -67.346, 101.151, -125.378, 47.884, 137.557]
  MoveL 288 to (320.19, 85.68, -150.19) mm, rotated rx -179.9 ry 0 rz -90 deg; joints [37.179, -67.459, 101.318, -125.463, 47.884, 137.646]
  MoveL 289 to (318, 85.6, -150.18) mm, rotated rx -179.9 ry 0 rz -90 deg; joints [37.11, -67.538, 101.438, -125.562, 47.861, 137.735]
  MoveL 290 to (315.96, 85.52, -150.95) mm, rotated rx -179.9 ry 0 rz -90 deg; joints [37.027, -67.574, 101.497, -125.661, 47.818, 137.815]
  MoveL 291 to (314.32, 85.45, -152.39) mm, rotated rx -179.9 ry 0 rz -90 deg; joints [36.94, -67.561, 101.486, -125.75, 47.761, 137.874]
  MoveL 292 to (313.31, 85.37, -154.33) mm, rotated rx -179.9 ry 0 rz -90 deg; joints [36.861, -67.501, 101.408, -125.816, 47.698, 137.907]
  MoveL 293 to (313.05, 85.29, -156.5) mm, rotated rx -179.9 ry 0 rz -90 deg; joints [36.801, -67.4, 101.273, -125.85, 47.637, 137.908]
  MoveL 294 to (313.58, 85.22, -158.62) mm, rotated rx -179.9 ry 0 rz -90 deg; joints [36.767, -67.273, 101.1, -125.85, 47.587, 137.879]
  MoveL 295 to (314.83, 85.14, -160.41) mm, rotated rx -179.9 ry 0 rz -90 deg; joints [36.764, -67.136, 100.91, -125.814, 47.555, 137.825]
  MoveL 296 to (316.64, 85.06, -161.64) mm, rotated rx -179.9 ry 0 rz -90 deg; joints [36.792, -67.006, 100.731, -125.749, 47.545, 137.751]
  MoveL 297 to (318.76, 84.99, -162.14) mm, rotated rx -179.9 ry 0 rz -90 deg; joints [36.848, -66.9, 100.585, -125.664, 47.559, 137.67]
  MoveL 298 to (320.93, 84.91, -161.86) mm, rotated rx -179.9 ry 0 rz -90 deg; joints [36.923, -66.832, 100.492, -125.57, 47.595, 137.593]
  MoveL 299 to (322.85, 84.83, -160.82) mm, rotated rx -179.9 ry 0 rz -90 deg; joints [37.009, -66.81, 100.464, -125.481, 47.65, 137.531]
  MoveL 300 to (324.28, 84.76, -159.16) mm, rotated rx -179.9 ry 0 rz -90 deg; joints [37.093, -66.837, 100.507, -125.408, 47.716, 137.493]
  MoveL 301 to (325.02, 84.68, -157.11) mm, rotated rx -179.9 ry 0 rz -90 deg; joints [37.166, -66.91, 100.614, -125.362, 47.786, 137.484]
  MoveL 302 to (324.98, 84.6, -154.92) mm, rotated rx -179.9 ry 0 rz -90 deg; joints [37.217, -67.017, 100.771, -125.348, 47.849, 137.506]
  MoveL 303 to (324.17, 84.53, -152.89) mm, rotated rx -179.9 ry 0 rz -90 deg; joints [37.241, -67.146, 100.959, -125.369, 47.899, 137.556]
  MoveL 304 to (322.68, 84.45, -151.29) mm, rotated rx -179.9 ry 0 rz -90 deg; joints [37.232, -67.279, 101.154, -125.422, 47.929, 137.629]
  MoveL 305 to (320.73, 84.37, -150.32) mm, rotated rx -179.9 ry 0 rz -90 deg; joints [37.194, -67.398, 101.329, -125.502, 47.936, 137.715]
  MoveL 306 to (318.55, 84.3, -150.11) mm, rotated rx -179.9 ry 0 rz -90 deg; joints [37.13, -67.487, 101.463, -125.598, 47.919, 137.806]
  MoveL 307 to (316.45, 84.22, -150.68) mm, rotated rx -179.9 ry 0 rz -90 deg; joints [37.049, -67.534, 101.538, -125.698, 47.88, 137.888]
  MoveL 308 to (314.68, 84.14, -151.97) mm, rotated rx -179.9 ry 0 rz -90 deg; joints [36.962, -67.534, 101.545, -125.791, 47.826, 137.954]
  MoveL 309 to (313.5, 84.07, -153.81) mm, rotated rx -179.9 ry 0 rz -90 deg; joints [36.88, -67.485, 101.483, -125.863, 47.764, 137.993]
  MoveL 310 to (313.04, 83.99, -155.95) mm, rotated rx -179.9 ry 0 rz -90 deg; joints [36.814, -67.393, 101.361, -125.906, 47.702, 138.003]
  MoveL 311 to (313.37, 83.91, -158.1) mm, rotated rx -179.9 ry 0 rz -90 deg; joints [36.774, -67.272, 101.195, -125.915, 47.648, 137.982]
  MoveL 312 to (314.45, 83.84, -160) mm, rotated rx -179.9 ry 0 rz -90 deg; joints [36.763, -67.135, 101.007, -125.888, 47.611, 137.933]
  MoveL 313 to (316.14, 83.76, -161.39) mm, rotated rx -179.9 ry 0 rz -90 deg; joints [36.783, -67.002, 100.823, -125.83, 47.595, 137.863]
  MoveL 314 to (318.21, 83.68, -162.09) mm, rotated rx -179.9 ry 0 rz -90 deg; joints [36.832, -66.889, 100.666, -125.748, 47.603, 137.783]
  MoveL 315 to (320.39, 83.61, -162) mm, rotated rx -179.9 ry 0 rz -90 deg; joints [36.904, -66.81, 100.558, -125.656, 47.634, 137.704]
  MoveL 316 to (322.4, 83.53, -161.14) mm, rotated rx -179.9 ry 0 rz -90 deg; joints [36.988, -66.776, 100.514, -125.564, 47.684, 137.637]
  MoveL 317 to (323.98, 83.45, -159.63) mm, rotated rx -179.9 ry 0 rz -90 deg; joints [37.073, -66.791, 100.539, -125.486, 47.748, 137.592]
  MoveL 318 to (324.9, 83.37, -157.65) mm, rotated rx -179.9 ry 0 rz -90 deg; joints [37.15, -66.853, 100.63, -125.432, 47.817, 137.575]
  MoveL 319 to (325.07, 83.3, -155.47) mm, rotated rx -179.9 ry 0 rz -90 deg; joints [37.208, -66.952, 100.777, -125.409, 47.883, 137.589]
  MoveL 320 to (324.44, 83.22, -153.38) mm, rotated rx -179.9 ry 0 rz -90 deg; joints [37.238, -67.077, 100.96, -125.422, 47.938, 137.633]
  MoveL 321 to (323.11, 83.14, -151.64) mm, rotated rx -179.9 ry 0 rz -90 deg; joints [37.238, -67.211, 101.155, -125.467, 47.973, 137.701]
  MoveL 322 to (321.25, 83.07, -150.49) mm, rotated rx -179.9 ry 0 rz -90 deg; joints [37.207, -67.334, 101.337, -125.541, 47.986, 137.785]
  MoveL 323 to (319.11, 82.99, -150.09) mm, rotated rx -179.9 ry 0 rz -90 deg; joints [37.149, -67.433, 101.483, -125.634, 47.975, 137.875]
  MoveL 324 to (316.96, 82.91, -150.47) mm, rotated rx -179.9 ry 0 rz -90 deg; joints [37.071, -67.491, 101.574, -125.735, 47.942, 137.961]
  MoveL 325 to (315.08, 82.84, -151.59) mm, rotated rx -179.9 ry 0 rz -90 deg; joints [36.985, -67.503, 101.599, -125.83, 47.891, 138.031]
  MoveL 326 to (313.73, 82.76, -153.31) mm, rotated rx -179.9 ry 0 rz -90 deg; joints [36.9, -67.466, 101.554, -125.909, 47.83, 138.078]
  MoveL 327 to (313.08, 82.68, -155.39) mm, rotated rx -179.9 ry 0 rz -90 deg; joints [36.83, -67.384, 101.446, -125.96, 47.767, 138.095]
  MoveL 328 to (313.21, 82.61, -157.57) mm, rotated rx -179.9 ry 0 rz -90 deg; joints [36.782, -67.269, 101.289, -125.978, 47.71, 138.082]
  MoveL 329 to (314.12, 82.53, -159.56) mm, rotated rx -179.9 ry 0 rz -90 deg; joints [36.763, -67.135, 101.104, -125.96, 47.668, 138.039]
  MoveL 330 to (315.67, 82.45, -161.1) mm, rotated rx -179.9 ry 0 rz -90 deg; joints [36.776, -66.999, 100.917, -125.909, 47.647, 137.974]
  MoveL 331 to (317.67, 82.38, -161.99) mm, rotated rx -179.9 ry 0 rz -90 deg; joints [36.818, -66.879, 100.751, -125.832, 47.648, 137.896]
  MoveL 332 to (319.85, 82.3, -162.1) mm, rotated rx -179.9 ry 0 rz -90 deg; joints [36.885, -66.791, 100.629, -125.741, 47.673, 137.815]
  MoveL 333 to (321.93, 82.22, -161.43) mm, rotated rx -179.9 ry 0 rz -90 deg; joints [36.966, -66.745, 100.568, -125.648, 47.719, 137.744]
  MoveL 334 to (323.63, 82.15, -160.06) mm, rotated rx -179.9 ry 0 rz -90 deg; joints [37.053, -66.748, 100.575, -125.565, 47.78, 137.693]
  MoveL 335 to (324.74, 82.07, -158.18) mm, rotated rx -179.9 ry 0 rz -90 deg; joints [37.133, -66.798, 100.651, -125.504, 47.849, 137.669]
  MoveL 336 to (325.1, 81.99, -156.02) mm, rotated rx -179.9 ry 0 rz -90 deg; joints [37.196, -66.889, 100.785, -125.473, 47.917, 137.675]
  MoveL 337 to (324.67, 81.92, -153.88) mm, rotated rx -179.9 ry 0 rz -90 deg; joints [37.234, -67.009, 100.96, -125.476, 47.975, 137.711]
  MoveL 338 to (323.51, 81.84, -152.03) mm, rotated rx -179.9 ry 0 rz -90 deg; joints [37.242, -67.142, 101.155, -125.514, 48.016, 137.774]
  MoveL 339 to (321.76, 81.76, -150.72) mm, rotated rx -179.9 ry 0 rz -90 deg; joints [37.218, -67.27, 101.343, -125.581, 48.035, 137.855]
  MoveL 340 to (319.66, 81.69, -150.11) mm, rotated rx -179.9 ry 0 rz -90 deg; joints [37.166, -67.376, 101.5, -125.67, 48.03, 137.944]
  MoveL 341 to (317.48, 81.61, -150.3) mm, rotated rx -179.9 ry 0 rz -90 deg; joints [37.093, -67.445, 101.606, -125.77, 48.002, 138.032]
  MoveL 342 to (315.51, 81.53, -151.24) mm, rotated rx -179.9 ry 0 rz -90 deg; joints [37.007, -67.469, 101.648, -125.868, 47.955, 138.107]
  MoveL 343 to (314.01, 81.46, -152.83) mm, rotated rx -179.9 ry 0 rz -90 deg; joints [36.921, -67.444, 101.62, -125.953, 47.896, 138.161]
  MoveL 344 to (313.17, 81.38, -154.85) mm, rotated rx -179.9 ry 0 rz -90 deg; joints [36.846, -67.373, 101.527, -126.012, 47.832, 138.186]
  MoveL 345 to (313.11, 81.3, -157.03) mm, rotated rx -179.9 ry 0 rz -90 deg; joints [36.792, -67.265, 101.381, -126.038, 47.774, 138.18]
  MoveL 346 to (313.82, 81.23, -159.09) mm, rotated rx -179.9 ry 0 rz -90 deg; joints [36.766, -67.134, 101.201, -126.029, 47.727, 138.144]
  MoveL 347 to (315.23, 81.15, -160.77) mm, rotated rx -179.9 ry 0 rz -90 deg; joints [36.77, -66.997, 101.012, -125.986, 47.7, 138.084]
  MoveL 348 to (317.13, 81.07, -161.83) mm, rotated rx -179.9 ry 0 rz -90 deg; joints [36.806, -66.872, 100.838, -125.915, 47.695, 138.008]
  MoveL 349 to (319.3, 81, -162.15) mm, rotated rx -179.9 ry 0 rz -90 deg; joints [36.867, -66.774, 100.704, -125.826, 47.714, 137.927]
  MoveL 350 to (321.43, 80.92, -161.67) mm, rotated rx -179.9 ry 0 rz -90 deg; joints [36.946, -66.717, 100.626, -125.732, 47.755, 137.852]
  MoveL 351 to (323.25, 80.84, -160.46) mm, rotated rx -179.9 ry 0 rz -90 deg; joints [37.032, -66.707, 100.615, -125.646, 47.813, 137.795]
  MoveL 352 to (324.53, 80.77, -158.69) mm, rotated rx -179.9 ry 0 rz -90 deg; joints [37.115, -66.746, 100.674, -125.578, 47.881, 137.764]
  MoveL 353 to (325.08, 80.69, -156.58) mm, rotated rx -179.9 ry 0 rz -90 deg; joints [37.183, -66.828, 100.795, -125.539, 47.95, 137.762]
  MoveL 354 to (324.85, 80.61, -154.4) mm, rotated rx -179.9 ry 0 rz -90 deg; joints [37.228, -66.942, 100.962, -125.533, 48.011, 137.791]
  MoveL 355 to (323.86, 80.54, -152.46) mm, rotated rx -179.9 ry 0 rz -90 deg; joints [37.243, -67.073, 101.154, -125.562, 48.057, 137.848]
  MoveL 356 to (322.24, 80.46, -150.99) mm, rotated rx -179.9 ry 0 rz -90 deg; joints [37.228, -67.203, 101.346, -125.623, 48.082, 137.925]
  MoveL 357 to (320.21, 80.38, -150.19) mm, rotated rx -179.9 ry 0 rz -90 deg; joints [37.182, -67.316, 101.513, -125.707, 48.083, 138.013]
  MoveL 358 to (318.02, 80.31, -150.18) mm, rotated rx -179.9 ry 0 rz -90 deg; joints [37.114, -67.396, 101.634, -125.806, 48.061, 138.103]
  MoveL 359 to (315.98, 80.23, -150.94) mm, rotated rx -179.9 ry 0 rz -90 deg; joints [37.03, -67.432, 101.693, -125.906, 48.018, 138.182]
  MoveL 360 to (314.33, 80.15, -152.38) mm, rotated rx -179.9 ry 0 rz -90 deg; joints [36.943, -67.419, 101.682, -125.994, 47.961, 138.241]
  MoveL 361 to (313.31, 80.08, -154.31) mm, rotated rx -179.9 ry 0 rz -90 deg; joints [36.864, -67.359, 101.605, -126.061, 47.898, 138.274]
  MoveL 362 to (313.05, 80, -156.48) mm, rotated rx -179.9 ry 0 rz -90 deg; joints [36.804, -67.259, 101.47, -126.096, 47.838, 138.276]
  MoveL 363 to (313.57, 79.92, -158.6) mm, rotated rx -179.9 ry 0 rz -90 deg; joints [36.77, -67.133, 101.297, -126.096, 47.788, 138.247]
  MoveL 364 to (314.82, 79.85, -160.4) mm, rotated rx -179.9 ry 0 rz -90 deg; joints [36.767, -66.996, 101.108, -126.061, 47.755, 138.193]
  MoveL 365 to (316.62, 79.77, -161.63) mm, rotated rx -179.9 ry 0 rz -90 deg; joints [36.795, -66.866, 100.928, -125.996, 47.744, 138.119]
  MoveL 366 to (318.74, 79.69, -162.14) mm, rotated rx -179.9 ry 0 rz -90 deg; joints [36.85, -66.76, 100.782, -125.911, 47.757, 138.039]
  MoveL 367 to (320.91, 79.62, -161.86) mm, rotated rx -179.9 ry 0 rz -90 deg; joints [36.925, -66.692, 100.688, -125.817, 47.793, 137.962]
  MoveL 368 to (322.84, 79.54, -160.83) mm, rotated rx -179.9 ry 0 rz -90 deg; joints [37.011, -66.67, 100.66, -125.727, 47.847, 137.899]
  MoveL 369 to (324.27, 79.46, -159.18) mm, rotated rx -179.9 ry 0 rz -90 deg; joints [37.095, -66.696, 100.702, -125.654, 47.913, 137.861]
  MoveL 370 to (325.02, 79.39, -157.13) mm, rotated rx -179.9 ry 0 rz -90 deg; joints [37.168, -66.768, 100.808, -125.607, 47.982, 137.851]
  MoveL 371 to (324.98, 79.31, -154.94) mm, rotated rx -179.9 ry 0 rz -90 deg; joints [37.22, -66.875, 100.965, -125.592, 48.046, 137.873]
  MoveL 372 to (324.18, 79.23, -152.91) mm, rotated rx -179.9 ry 0 rz -90 deg; joints [37.243, -67.003, 101.153, -125.613, 48.096, 137.923]
  MoveL 373 to (322.7, 79.16, -151.3) mm, rotated rx -179.9 ry 0 rz -90 deg; joints [37.235, -67.136, 101.348, -125.666, 48.127, 137.996]
  MoveL 374 to (320.75, 79.08, -150.32) mm, rotated rx -179.9 ry 0 rz -90 deg; joints [37.197, -67.255, 101.523, -125.745, 48.135, 138.082]
  MoveL 375 to (318.57, 79, -150.11) mm, rotated rx -179.9 ry 0 rz -90 deg; joints [37.133, -67.344, 101.657, -125.841, 48.118, 138.172]
  MoveL 376 to (316.46, 78.93, -150.68) mm, rotated rx -179.9 ry 0 rz -90 deg; joints [37.053, -67.392, 101.733, -125.942, 48.08, 138.255]
  MoveL 377 to (314.7, 78.85, -151.96) mm, rotated rx -179.9 ry 0 rz -90 deg; joints [36.965, -67.391, 101.74, -126.035, 48.027, 138.32]
  MoveL 378 to (313.5, 78.77, -153.79) mm, rotated rx -179.9 ry 0 rz -90 deg; joints [36.883, -67.343, 101.679, -126.107, 47.965, 138.36]
  MoveL 379 to (313.04, 78.69, -155.93) mm, rotated rx -179.9 ry 0 rz -90 deg; joints [36.818, -67.252, 101.558, -126.151, 47.903, 138.37]
  MoveL 380 to (313.37, 78.62, -158.09) mm, rotated rx -179.9 ry 0 rz -90 deg; joints [36.776, -67.131, 101.392, -126.16, 47.849, 138.349]
  MoveL 381 to (314.44, 78.54, -159.99) mm, rotated rx -179.9 ry 0 rz -90 deg; joints [36.765, -66.995, 101.204, -126.134, 47.811, 138.3]
  MoveL 382 to (316.12, 78.46, -161.38) mm, rotated rx -179.9 ry 0 rz -90 deg; joints [36.786, -66.861, 101.02, -126.076, 47.794, 138.231]
  MoveL 383 to (318.19, 78.39, -162.09) mm, rotated rx -179.9 ry 0 rz -90 deg; joints [36.834, -66.748, 100.863, -125.995, 47.801, 138.151]
  MoveL 384 to (320.38, 78.31, -162.01) mm, rotated rx -179.9 ry 0 rz -90 deg; joints [36.905, -66.67, 100.754, -125.902, 47.832, 138.072]
  MoveL 385 to (322.39, 78.23, -161.15) mm, rotated rx -179.9 ry 0 rz -90 deg; joints [36.989, -66.635, 100.709, -125.81, 47.881, 138.005]
  MoveL 386 to (323.96, 78.16, -159.64) mm, rotated rx -179.9 ry 0 rz -90 deg; joints [37.075, -66.65, 100.733, -125.731, 47.945, 137.959]
  MoveL 387 to (324.9, 78.08, -157.67) mm, rotated rx -179.9 ry 0 rz -90 deg; joints [37.152, -66.711, 100.824, -125.677, 48.014, 137.942]
  MoveL 388 to (325.07, 78, -155.49) mm, rotated rx -179.9 ry 0 rz -90 deg; joints [37.21, -66.81, 100.971, -125.654, 48.08, 137.956]
  MoveL 389 to (324.45, 77.93, -153.39) mm, rotated rx -179.9 ry 0 rz -90 deg; joints [37.241, -66.934, 101.153, -125.665, 48.135, 137.999]
  MoveL 390 to (323.13, 77.85, -151.65) mm, rotated rx -179.9 ry 0 rz -90 deg; joints [37.241, -67.067, 101.348, -125.71, 48.171, 138.067]
  MoveL 391 to (321.27, 77.77, -150.5) mm, rotated rx -179.9 ry 0 rz -90 deg; joints [37.21, -67.191, 101.531, -125.784, 48.185, 138.151]
  MoveL 392 to (319.13, 77.7, -150.09) mm, rotated rx -179.9 ry 0 rz -90 deg; joints [37.152, -67.289, 101.677, -125.876, 48.174, 138.241]
  MoveL 393 to (316.97, 77.62, -150.46) mm, rotated rx -179.9 ry 0 rz -90 deg; joints [37.075, -67.348, 101.769, -125.977, 48.142, 138.327]
  MoveL 394 to (315.1, 77.54, -151.58) mm, rotated rx -179.9 ry 0 rz -90 deg; joints [36.988, -67.36, 101.794, -126.073, 48.092, 138.397]
  MoveL 395 to (313.74, 77.47, -153.29) mm, rotated rx -179.9 ry 0 rz -90 deg; joints [36.904, -67.324, 101.749, -126.152, 48.031, 138.444]
  MoveL 396 to (313.08, 77.39, -155.37) mm, rotated rx -179.9 ry 0 rz -90 deg; joints [36.833, -67.242, 101.642, -126.204, 47.968, 138.462]
  MoveL 397 to (313.21, 77.31, -157.56) mm, rotated rx -179.9 ry 0 rz -90 deg; joints [36.785, -67.128, 101.485, -126.222, 47.911, 138.448]
  MoveL 398 to (314.11, 77.24, -159.55) mm, rotated rx -179.9 ry 0 rz -90 deg; joints [36.766, -66.994, 101.301, -126.204, 47.869, 138.406]
  MoveL 399 to (315.65, 77.16, -161.09) mm, rotated rx -179.9 ry 0 rz -90 deg; joints [36.778, -66.858, 101.113, -126.154, 47.846, 138.341]
  MoveL 400 to (317.65, 77.08, -161.98) mm, rotated rx -179.9 ry 0 rz -90 deg; joints [36.82, -66.738, 100.947, -126.078, 47.847, 138.262]
  MoveL 401 to (319.83, 77.01, -162.1) mm, rotated rx -179.9 ry 0 rz -90 deg; joints [36.887, -66.65, 100.825, -125.986, 47.872, 138.182]
  MoveL 402 to (321.91, 76.93, -161.44) mm, rotated rx -179.9 ry 0 rz -90 deg; joints [36.968, -66.604, 100.762, -125.893, 47.917, 138.111]
  MoveL 403 to (323.62, 76.85, -160.08) mm, rotated rx -179.9 ry 0 rz -90 deg; joints [37.055, -66.606, 100.769, -125.81, 47.978, 138.06]
  MoveL 404 to (324.73, 76.78, -158.2) mm, rotated rx -179.9 ry 0 rz -90 deg; joints [37.135, -66.656, 100.844, -125.748, 48.046, 138.035]
  MoveL 405 to (325.1, 76.7, -156.04) mm, rotated rx -179.9 ry 0 rz -90 deg; joints [37.198, -66.746, 100.978, -125.717, 48.114, 138.041]
  MoveL 406 to (324.68, 76.62, -153.9) mm, rotated rx -179.9 ry 0 rz -90 deg; joints [37.236, -66.866, 101.153, -125.719, 48.172, 138.077]
  MoveL 407 to (323.52, 76.55, -152.05) mm, rotated rx -179.9 ry 0 rz -90 deg; joints [37.245, -66.998, 101.347, -125.756, 48.214, 138.139]
  MoveL 408 to (321.78, 76.47, -150.73) mm, rotated rx -179.9 ry 0 rz -90 deg; joints [37.221, -67.126, 101.535, -125.823, 48.233, 138.22]
  MoveL 409 to (319.68, 76.39, -150.12) mm, rotated rx -179.9 ry 0 rz -90 deg; joints [37.17, -67.232, 101.693, -125.912, 48.229, 138.31]
  MoveL 410 to (317.5, 76.32, -150.29) mm, rotated rx -179.9 ry 0 rz -90 deg; joints [37.096, -67.301, 101.8, -126.012, 48.202, 138.397]
  MoveL 411 to (315.53, 76.24, -151.23) mm, rotated rx -179.9 ry 0 rz -90 deg; joints [37.011, -67.326, 101.842, -126.111, 48.156, 138.473]
  MoveL 412 to (314.02, 76.16, -152.81) mm, rotated rx -179.9 ry 0 rz -90 deg; joints [36.925, -67.301, 101.815, -126.195, 48.097, 138.526]
  MoveL 413 to (313.18, 76.09, -154.83) mm, rotated rx -179.9 ry 0 rz -90 deg; joints [36.85, -67.231, 101.722, -126.255, 48.034, 138.551]
  MoveL 414 to (313.1, 76.01, -157.01) mm, rotated rx -179.9 ry 0 rz -90 deg; joints [36.795, -67.123, 101.577, -126.282, 47.975, 138.546]
  MoveL 415 to (313.81, 75.93, -159.08) mm, rotated rx -179.9 ry 0 rz -90 deg; joints [36.768, -66.992, 101.397, -126.273, 47.928, 138.51]
  MoveL 416 to (315.21, 75.86, -160.76) mm, rotated rx -179.9 ry 0 rz -90 deg; joints [36.773, -66.856, 101.208, -126.23, 47.9, 138.45]
  MoveL 417 to (317.12, 75.78, -161.83) mm, rotated rx -179.9 ry 0 rz -90 deg; joints [36.808, -66.73, 101.034, -126.159, 47.895, 138.374]
  MoveL 418 to (319.28, 75.7, -162.15) mm, rotated rx -179.9 ry 0 rz -90 deg; joints [36.869, -66.633, 100.899, -126.071, 47.913, 138.293]
  MoveL 419 to (321.41, 75.63, -161.68) mm, rotated rx -179.9 ry 0 rz -90 deg; joints [36.947, -66.575, 100.82, -125.977, 47.954, 138.219]
  MoveL 420 to (323.24, 75.55, -160.48) mm, rotated rx -179.9 ry 0 rz -90 deg; joints [37.034, -66.565, 100.809, -125.89, 48.011, 138.161]
  MoveL 421 to (324.52, 75.47, -158.71) mm, rotated rx -179.9 ry 0 rz -90 deg; joints [37.117, -66.603, 100.867, -125.822, 48.078, 138.13]
  MoveL 422 to (325.08, 75.4, -156.59) mm, rotated rx -179.9 ry 0 rz -90 deg; joints [37.185, -66.684, 100.988, -125.782, 48.147, 138.128]
  MoveL 423 to (324.86, 75.32, -154.42) mm, rotated rx -179.9 ry 0 rz -90 deg; joints [37.23, -66.798, 101.155, -125.776, 48.208, 138.157]
  MoveL 424 to (323.87, 75.24, -152.47) mm, rotated rx -179.9 ry 0 rz -90 deg; joints [37.246, -66.929, 101.346, -125.804, 48.255, 138.213]
  MoveL 425 to (322.26, 75.17, -151) mm, rotated rx -179.9 ry 0 rz -90 deg; joints [37.231, -67.059, 101.538, -125.864, 48.28, 138.29]
  MoveL 426 to (320.23, 75.09, -150.2) mm, rotated rx -179.9 ry 0 rz -90 deg; joints [37.186, -67.172, 101.706, -125.949, 48.282, 138.378]
  MoveL 427 to (318.04, 75.01, -150.17) mm, rotated rx -179.9 ry 0 rz -90 deg; joints [37.117, -67.252, 101.827, -126.047, 48.261, 138.467]
  MoveL 428 to (315.99, 74.94, -150.93) mm, rotated rx -179.9 ry 0 rz -90 deg; joints [37.034, -67.288, 101.886, -126.147, 48.219, 138.546]
  MoveL 429 to (314.35, 74.86, -152.36) mm, rotated rx -179.9 ry 0 rz -90 deg; joints [36.947, -67.276, 101.877, -126.236, 48.163, 138.606]
  MoveL 430 to (313.32, 74.78, -154.29) mm, rotated rx -179.9 ry 0 rz -90 deg; joints [36.868, -67.216, 101.8, -126.303, 48.1, 138.639]
  MoveL 431 to (313.05, 74.71, -156.46) mm, rotated rx -179.9 ry 0 rz -90 deg; joints [36.807, -67.117, 101.666, -126.339, 48.039, 138.641]
  MoveL 432 to (313.56, 74.63, -158.58) mm, rotated rx -179.9 ry 0 rz -90 deg; joints [36.773, -66.991, 101.492, -126.339, 47.989, 138.612]
  MoveL 433 to (314.8, 74.55, -160.38) mm, rotated rx -179.9 ry 0 rz -90 deg; joints [36.769, -66.854, 101.303, -126.304, 47.955, 138.558]
  MoveL 434 to (316.6, 74.48, -161.62) mm, rotated rx -179.9 ry 0 rz -90 deg; joints [36.797, -66.724, 101.123, -126.24, 47.944, 138.485]
  MoveL 435 to (318.72, 74.4, -162.14) mm, rotated rx -179.9 ry 0 rz -90 deg; joints [36.852, -66.618, 100.976, -126.155, 47.956, 138.404]
  MoveL 436 to (320.89, 74.32, -161.87) mm, rotated rx -179.9 ry 0 rz -90 deg; joints [36.927, -66.55, 100.882, -126.061, 47.991, 138.327]
  MoveL 437 to (322.82, 74.25, -160.84) mm, rotated rx -179.9 ry 0 rz -90 deg; joints [37.013, -66.527, 100.853, -125.971, 48.045, 138.265]
  MoveL 438 to (324.26, 74.17, -159.19) mm, rotated rx -179.9 ry 0 rz -90 deg; joints [37.097, -66.553, 100.895, -125.897, 48.11, 138.226]
  MoveL 439 to (325.01, 74.09, -157.14) mm, rotated rx -179.9 ry 0 rz -90 deg; joints [37.17, -66.625, 101, -125.85, 48.18, 138.216]
  MoveL 440 to (324.99, 74.01, -154.96) mm, rotated rx -179.9 ry 0 rz -90 deg; joints [37.222, -66.731, 101.157, -125.834, 48.244, 138.237]
  MoveL 441 to (324.19, 73.94, -152.93) mm, rotated rx -179.9 ry 0 rz -90 deg; joints [37.246, -66.859, 101.345, -125.854, 48.295, 138.287]
  MoveL 442 to (322.72, 73.86, -151.31) mm, rotated rx -179.9 ry 0 rz -90 deg; joints [37.238, -66.991, 101.539, -125.907, 48.326, 138.36]
  MoveL 443 to (320.76, 73.78, -150.33) mm, rotated rx -179.9 ry 0 rz -90 deg; joints [37.2, -67.11, 101.715, -125.986, 48.334, 138.446]
  MoveL 444 to (318.59, 73.71, -150.1) mm, rotated rx -179.9 ry 0 rz -90 deg; joints [37.137, -67.199, 101.85, -126.082, 48.318, 138.536]
  MoveL 445 to (316.48, 73.63, -150.67) mm, rotated rx -179.9 ry 0 rz -90 deg; joints [37.056, -67.247, 101.926, -126.182, 48.281, 138.619]
  MoveL 446 to (314.71, 73.55, -151.95) mm, rotated rx -179.9 ry 0 rz -90 deg; joints [36.969, -67.247, 101.934, -126.276, 48.228, 138.684]
  MoveL 447 to (313.51, 73.48, -153.77) mm, rotated rx -179.9 ry 0 rz -90 deg; joints [36.887, -67.199, 101.873, -126.349, 48.166, 138.724]
  MoveL 448 to (313.04, 73.4, -155.91) mm, rotated rx -179.9 ry 0 rz -90 deg; joints [36.821, -67.109, 101.752, -126.393, 48.104, 138.734]
  MoveL 449 to (313.36, 73.32, -158.07) mm, rotated rx -179.9 ry 0 rz -90 deg; joints [36.779, -66.988, 101.587, -126.403, 48.051, 138.713]
  MoveL 450 to (314.43, 73.25, -159.97) mm, rotated rx -179.9 ry 0 rz -90 deg; joints [36.768, -66.852, 101.399, -126.377, 48.012, 138.665]
  MoveL 451 to (316.11, 73.17, -161.37) mm, rotated rx -179.9 ry 0 rz -90 deg; joints [36.788, -66.719, 101.214, -126.319, 47.995, 138.595]
  MoveL 452 to (318.17, 73.09, -162.08) mm, rotated rx -179.9 ry 0 rz -90 deg; joints [36.837, -66.606, 101.057, -126.238, 48.001, 138.515]
  MoveL 453 to (320.36, 73.02, -162.01) mm, rotated rx -179.9 ry 0 rz -90 deg; joints [36.907, -66.527, 100.948, -126.145, 48.03, 138.436]
  MoveL 454 to (322.37, 72.94, -161.17) mm, rotated rx -179.9 ry 0 rz -90 deg; joints [36.991, -66.493, 100.902, -126.053, 48.08, 138.369]
  MoveL 455 to (323.95, 72.86, -159.66) mm, rotated rx -179.9 ry 0 rz -90 deg; joints [37.077, -66.506, 100.926, -125.974, 48.143, 138.324]
  MoveL 456 to (324.89, 72.79, -157.69) mm, rotated rx -179.9 ry 0 rz -90 deg; joints [37.154, -66.567, 101.016, -125.919, 48.212, 138.307]
  MoveL 457 to (325.07, 72.71, -155.51) mm, rotated rx -179.9 ry 0 rz -90 deg; joints [37.212, -66.666, 101.162, -125.895, 48.278, 138.32]
  MoveL 458 to (324.46, 72.63, -153.41) mm, rotated rx -179.9 ry 0 rz -90 deg; joints [37.243, -66.789, 101.344, -125.906, 48.333, 138.363]
  MoveL 459 to (323.14, 72.56, -151.67) mm, rotated rx -179.9 ry 0 rz -90 deg; joints [37.244, -66.922, 101.539, -125.951, 48.37, 138.431]
  MoveL 460 to (321.29, 72.48, -150.51) mm, rotated rx -179.9 ry 0 rz -90 deg; joints [37.213, -67.046, 101.722, -126.024, 48.384, 138.514]
  MoveL 461 to (319.14, 72.4, -150.09) mm, rotated rx -179.9 ry 0 rz -90 deg; joints [37.155, -67.144, 101.869, -126.116, 48.375, 138.605]
  MoveL 462 to (316.99, 72.33, -150.45) mm, rotated rx -179.9 ry 0 rz -90 deg; joints [37.078, -67.203, 101.961, -126.217, 48.343, 138.69]
  MoveL 463 to (315.11, 72.25, -151.57) mm, rotated rx -179.9 ry 0 rz -90 deg; joints [36.992, -67.215, 101.986, -126.314, 48.293, 138.761]
  MoveL 464 to (313.75, 72.17, -153.27) mm, rotated rx -179.9 ry 0 rz -90 deg; joints [36.907, -67.179, 101.943, -126.393, 48.233, 138.807]
  MoveL 465 to (313.08, 72.1, -155.36) mm, rotated rx -179.9 ry 0 rz -90 deg; joints [36.836, -67.099, 101.835, -126.445, 48.17, 138.825]
  MoveL 466 to (313.2, 72.02, -157.54) mm, rotated rx -179.9 ry 0 rz -90 deg; joints [36.788, -66.984, 101.679, -126.464, 48.113, 138.812]
  MoveL 467 to (314.1, 71.94, -159.53) mm, rotated rx -179.9 ry 0 rz -90 deg; joints [36.769, -66.851, 101.495, -126.447, 48.071, 138.77]
  MoveL 468 to (315.64, 71.87, -161.08) mm, rotated rx -179.9 ry 0 rz -90 deg; joints [36.781, -66.715, 101.307, -126.396, 48.047, 138.705]
  MoveL 469 to (317.63, 71.79, -161.98) mm, rotated rx -179.9 ry 0 rz -90 deg; joints [36.823, -66.596, 101.141, -126.32, 48.047, 138.627]
  MoveL 470 to (319.81, 71.71, -162.1) mm, rotated rx -179.9 ry 0 rz -90 deg; joints [36.889, -66.507, 101.018, -126.229, 48.071, 138.546]
  MoveL 471 to (321.89, 71.64, -161.45) mm, rotated rx -179.9 ry 0 rz -90 deg; joints [36.97, -66.461, 100.955, -126.135, 48.116, 138.475]
  MoveL 472 to (323.61, 71.56, -160.09) mm, rotated rx -179.9 ry 0 rz -90 deg; joints [37.057, -66.462, 100.961, -126.052, 48.176, 138.424]
  MoveL 473 to (324.73, 71.48, -158.21) mm, rotated rx -179.9 ry 0 rz -90 deg; joints [37.137, -66.512, 101.036, -125.99, 48.244, 138.399]
  MoveL 474 to (325.1, 71.41, -156.06) mm, rotated rx -179.9 ry 0 rz -90 deg; joints [37.2, -66.602, 101.169, -125.958, 48.312, 138.404]
  MoveL 475 to (324.68, 71.33, -153.92) mm, rotated rx -179.9 ry 0 rz -90 deg; joints [37.239, -66.72, 101.344, -125.96, 48.37, 138.44]
  MoveL 476 to (323.53, 71.25, -152.06) mm, rotated rx -179.9 ry 0 rz -90 deg; joints [37.247, -66.852, 101.538, -125.996, 48.413, 138.502]
  MoveL 477 to (321.79, 71.18, -150.74) mm, rotated rx -179.9 ry 0 rz -90 deg; joints [37.224, -66.98, 101.726, -126.063, 48.433, 138.583]
  MoveL 478 to (319.7, 71.1, -150.12) mm, rotated rx -179.9 ry 0 rz -90 deg; joints [37.173, -67.086, 101.884, -126.152, 48.43, 138.672]
  MoveL 479 to (317.52, 71.02, -150.29) mm, rotated rx -179.9 ry 0 rz -90 deg; joints [37.1, -67.156, 101.991, -126.252, 48.403, 138.76]
  MoveL 480 to (315.54, 70.95, -151.22) mm, rotated rx -179.9 ry 0 rz -90 deg; joints [37.014, -67.18, 102.034, -126.35, 48.357, 138.835]
  MoveL 481 to (314.03, 70.87, -152.8) mm, rotated rx -179.9 ry 0 rz -90 deg; joints [36.928, -67.156, 102.008, -126.435, 48.299, 138.889]
  MoveL 482 to (313.18, 70.79, -154.81) mm, rotated rx -179.9 ry 0 rz -90 deg; joints [36.853, -67.086, 101.915, -126.495, 48.236, 138.914]
  MoveL 483 to (313.1, 70.72, -156.99) mm, rotated rx -179.9 ry 0 rz -90 deg; joints [36.798, -66.979, 101.77, -126.523, 48.177, 138.909]
  MoveL 484 to (313.8, 70.64, -159.06) mm, rotated rx -179.9 ry 0 rz -90 deg; joints [36.771, -66.849, 101.591, -126.514, 48.13, 138.873]
  MoveL 485 to (315.2, 70.56, -160.74) mm, rotated rx -179.9 ry 0 rz -90 deg; joints [36.775, -66.712, 101.401, -126.472, 48.101, 138.813]
  MoveL 486 to (317.1, 70.49, -161.82) mm, rotated rx -179.9 ry 0 rz -90 deg; joints [36.81, -66.587, 101.227, -126.401, 48.095, 138.737]
  MoveL 487 to (319.26, 70.41, -162.15) mm, rotated rx -179.9 ry 0 rz -90 deg; joints [36.871, -66.49, 101.091, -126.313, 48.113, 138.656]
  MoveL 488 to (321.39, 70.33, -161.68) mm, rotated rx -179.9 ry 0 rz -90 deg; joints [36.949, -66.432, 101.012, -126.219, 48.153, 138.582]
  MoveL 489 to (323.22, 70.26, -160.49) mm, rotated rx -179.9 ry 0 rz -90 deg; joints [37.036, -66.421, 101.001, -126.131, 48.209, 138.525]
  MoveL 490 to (324.51, 70.18, -158.72) mm, rotated rx -179.9 ry 0 rz -90 deg; joints [37.119, -66.459, 101.058, -126.063, 48.276, 138.493]
  MoveL 491 to (325.08, 70.1, -156.61) mm, rotated rx -179.9 ry 0 rz -90 deg; joints [37.187, -66.539, 101.178, -126.023, 48.345, 138.491]
  MoveL 492 to (324.86, 70.03, -154.44) mm, rotated rx -179.9 ry 0 rz -90 deg; joints [37.233, -66.652, 101.345, -126.016, 48.407, 138.519]
  MoveL 493 to (323.88, 69.95, -152.49) mm, rotated rx -179.9 ry 0 rz -90 deg; joints [37.249, -66.782, 101.536, -126.044, 48.454, 138.575]
  MoveL 494 to (322.28, 69.87, -151.01) mm, rotated rx -179.9 ry 0 rz -90 deg; joints [37.234, -66.913, 101.728, -126.103, 48.48, 138.652]
  MoveL 495 to (320.25, 69.8, -150.2) mm, rotated rx -179.9 ry 0 rz -90 deg; joints [37.189, -67.025, 101.896, -126.187, 48.483, 138.74]
  MoveL 496 to (318.06, 69.72, -150.17) mm, rotated rx -179.9 ry 0 rz -90 deg; joints [37.12, -67.105, 102.018, -126.286, 48.462, 138.829]
  MoveL 497 to (316.01, 69.64, -150.92) mm, rotated rx -179.9 ry 0 rz -90 deg; joints [37.037, -67.142, 102.078, -126.386, 48.421, 138.908]
  MoveL 498 to (314.36, 69.56, -152.35) mm, rotated rx -179.9 ry 0 rz -90 deg; joints [36.95, -67.13, 102.069, -126.475, 48.365, 138.968]
  MoveL 499 to (313.32, 69.49, -154.27) mm, rotated rx -179.9 ry 0 rz -90 deg; joints [36.871, -67.071, 101.992, -126.542, 48.303, 139.001]
  MoveL 500 to (313.04, 69.41, -156.44) mm, rotated rx -179.9 ry 0 rz -90 deg; joints [36.81, -66.972, 101.858, -126.579, 48.242, 139.003]
  MoveL 501 to (313.56, 69.33, -158.57) mm, rotated rx -179.9 ry 0 rz -90 deg; joints [36.776, -66.846, 101.685, -126.58, 48.191, 138.975]
  MoveL 502 to (314.79, 69.26, -160.37) mm, rotated rx -179.9 ry 0 rz -90 deg; joints [36.772, -66.71, 101.496, -126.545, 48.157, 138.921]
  MoveL 503 to (316.58, 69.18, -161.61) mm, rotated rx -179.9 ry 0 rz -90 deg; joints [36.799, -66.58, 101.316, -126.481, 48.145, 138.848]
  MoveL 504 to (318.71, 69.1, -162.14) mm, rotated rx -179.9 ry 0 rz -90 deg; joints [36.854, -66.475, 101.168, -126.396, 48.157, 138.767]
  MoveL 505 to (320.87, 69.03, -161.87) mm, rotated rx -179.9 ry 0 rz -90 deg; joints [36.929, -66.406, 101.074, -126.302, 48.191, 138.69]
  MoveL 506 to (322.81, 68.95, -160.85) mm, rotated rx -179.9 ry 0 rz -90 deg; joints [37.015, -66.383, 101.045, -126.212, 48.244, 138.627]
  MoveL 507 to (324.25, 68.87, -159.21) mm, rotated rx -179.9 ry 0 rz -90 deg; joints [37.099, -66.409, 101.085, -126.138, 48.309, 138.588]
  MoveL 508 to (325.01, 68.8, -157.16) mm, rotated rx -179.9 ry 0 rz -90 deg; joints [37.172, -66.479, 101.19, -126.089, 48.378, 138.579]
  MoveL 509 to (324.99, 68.72, -154.98) mm, rotated rx -179.9 ry 0 rz -90 deg; joints [37.224, -66.585, 101.347, -126.074, 48.442, 138.599]
  MoveL 510 to (324.2, 68.64, -152.94) mm, rotated rx -179.9 ry 0 rz -90 deg; joints [37.248, -66.712, 101.535, -126.093, 48.494, 138.649]
  MoveL 511 to (322.73, 68.57, -151.32) mm, rotated rx -179.9 ry 0 rz -90 deg; joints [37.241, -66.844, 101.729, -126.145, 48.526, 138.721]
  MoveL 512 to (320.78, 68.49, -150.33) mm, rotated rx -179.9 ry 0 rz -90 deg; joints [37.203, -66.963, 101.905, -126.224, 48.535, 138.808]
  MoveL 513 to (318.61, 68.41, -150.1) mm, rotated rx -179.9 ry 0 rz -90 deg; joints [37.14, -67.052, 102.04, -126.32, 48.52, 138.898]
  MoveL 514 to (316.5, 68.34, -150.66) mm, rotated rx -179.9 ry 0 rz -90 deg; joints [37.059, -67.1, 102.116, -126.421, 48.483, 138.98]
  MoveL 515 to (314.72, 68.26, -151.93) mm, rotated rx -179.9 ry 0 rz -90 deg; joints [36.972, -67.101, 102.125, -126.514, 48.431, 139.046]
  MoveL 516 to (313.52, 68.18, -153.76) mm, rotated rx -179.9 ry 0 rz -90 deg; joints [36.89, -67.053, 102.065, -126.588, 48.369, 139.086]
  MoveL 517 to (313.04, 68.11, -155.89) mm, rotated rx -179.9 ry 0 rz -90 deg; joints [36.824, -66.963, 101.944, -126.632, 48.307, 139.096]
  MoveL 518 to (313.35, 68.03, -158.05) mm, rotated rx -179.9 ry 0 rz -90 deg; joints [36.782, -66.843, 101.779, -126.642, 48.253, 139.075]
  MoveL 519 to (314.42, 67.95, -159.96) mm, rotated rx -179.9 ry 0 rz -90 deg; joints [36.771, -66.708, 101.592, -126.617, 48.214, 139.027]
  MoveL 520 to (316.09, 67.88, -161.36) mm, rotated rx -179.9 ry 0 rz -90 deg; joints [36.79, -66.575, 101.407, -126.559, 48.196, 138.957]
  MoveL 521 to (318.15, 67.8, -162.08) mm, rotated rx -179.9 ry 0 rz -90 deg; joints [36.839, -66.462, 101.249, -126.479, 48.202, 138.878]
  MoveL 522 to (320.34, 67.72, -162.01) mm, rotated rx -179.9 ry 0 rz -90 deg; joints [36.909, -66.383, 101.139, -126.386, 48.23, 138.799]
  MoveL 523 to (322.36, 67.65, -161.18) mm, rotated rx -179.9 ry 0 rz -90 deg; joints [36.993, -66.348, 101.093, -126.293, 48.279, 138.731]
  MoveL 524 to (323.94, 67.57, -159.67) mm, rotated rx -179.9 ry 0 rz -90 deg; joints [37.079, -66.361, 101.116, -126.214, 48.342, 138.686]
  MoveL 525 to (324.89, 67.49, -157.7) mm, rotated rx -179.9 ry 0 rz -90 deg; joints [37.156, -66.421, 101.206, -126.158, 48.411, 138.668]
  MoveL 526 to (325.07, 67.42, -155.53) mm, rotated rx -179.9 ry 0 rz -90 deg; joints [37.214, -66.519, 101.351, -126.134, 48.477, 138.682]
  MoveL 527 to (324.47, 67.34, -153.43) mm, rotated rx -179.9 ry 0 rz -90 deg; joints [37.246, -66.643, 101.533, -126.144, 48.532, 138.724]
  MoveL 528 to (323.15, 67.26, -151.68) mm, rotated rx -179.9 ry 0 rz -90 deg; joints [37.247, -66.775, 101.728, -126.188, 48.57, 138.792]
  MoveL 529 to (321.31, 67.19, -150.52) mm, rotated rx -179.9 ry 0 rz -90 deg; joints [37.216, -66.898, 101.911, -126.261, 48.585, 138.875]
  MoveL 530 to (319.16, 67.11, -150.09) mm, rotated rx -179.9 ry 0 rz -90 deg; joints [37.159, -66.996, 102.058, -126.354, 48.576, 138.965]
  MoveL 531 to (317.01, 67.03, -150.45) mm, rotated rx -179.9 ry 0 rz -90 deg; joints [37.082, -67.056, 102.151, -126.455, 48.545, 139.051]
  MoveL 532 to (315.12, 66.96, -151.55) mm, rotated rx -179.9 ry 0 rz -90 deg; joints [36.995, -67.069, 102.177, -126.551, 48.496, 139.121]
  MoveL 533 to (313.76, 66.88, -153.26) mm, rotated rx -179.9 ry 0 rz -90 deg; joints [36.91, -67.033, 102.134, -126.631, 48.436, 139.168]
  MoveL 534 to (313.09, 66.8, -155.34) mm, rotated rx -179.9 ry 0 rz -90 deg; joints [36.839, -66.953, 102.027, -126.684, 48.373, 139.186]
  MoveL 535 to (313.2, 66.73, -157.52) mm, rotated rx -179.9 ry 0 rz -90 deg; joints [36.791, -66.839, 101.871, -126.703, 48.316, 139.173]
  MoveL 536 to (314.08, 66.65, -159.52) mm, rotated rx -179.9 ry 0 rz -90 deg; joints [36.771, -66.706, 101.687, -126.686, 48.273, 139.131]
  MoveL 537 to (315.62, 66.57, -161.07) mm, rotated rx -179.9 ry 0 rz -90 deg; joints [36.783, -66.571, 101.499, -126.636, 48.249, 139.066]
  MoveL 538 to (317.61, 66.5, -161.97) mm, rotated rx -179.9 ry 0 rz -90 deg; joints [36.825, -66.451, 101.332, -126.56, 48.248, 138.988]
  MoveL 539 to (319.79, 66.42, -162.11) mm, rotated rx -179.9 ry 0 rz -90 deg; joints [36.891, -66.362, 101.209, -126.469, 48.271, 138.908]
  MoveL 540 to (321.88, 66.34, -161.46) mm, rotated rx -179.9 ry 0 rz -90 deg; joints [36.972, -66.316, 101.145, -126.375, 48.315, 138.837]
  MoveL 541 to (323.6, 66.27, -160.1) mm, rotated rx -179.9 ry 0 rz -90 deg; joints [37.059, -66.317, 101.151, -126.291, 48.375, 138.785]
  MoveL 542 to (324.72, 66.19, -158.23) mm, rotated rx -179.9 ry 0 rz -90 deg; joints [37.139, -66.365, 101.225, -126.229, 48.443, 138.76]
  MoveL 543 to (325.1, 66.11, -156.08) mm, rotated rx -179.9 ry 0 rz -90 deg; joints [37.203, -66.455, 101.357, -126.196, 48.511, 138.765]
  MoveL 544 to (324.69, 66.04, -153.93) mm, rotated rx -179.9 ry 0 rz -90 deg; joints [37.241, -66.573, 101.532, -126.197, 48.57, 138.801]
  MoveL 545 to (323.54, 65.96, -152.07) mm, rotated rx -179.9 ry 0 rz -90 deg; joints [37.25, -66.705, 101.726, -126.233, 48.612, 138.863]
  MoveL 546 to (321.81, 65.88, -150.74) mm, rotated rx -179.9 ry 0 rz -90 deg; joints [37.227, -66.832, 101.915, -126.3, 48.634, 138.943]
  MoveL 547 to (319.72, 65.81, -150.12) mm, rotated rx -179.9 ry 0 rz -90 deg; joints [37.176, -66.938, 102.073, -126.388, 48.631, 139.033]
  MoveL 548 to (317.54, 65.73, -150.28) mm, rotated rx -179.9 ry 0 rz -90 deg; joints [37.103, -67.008, 102.181, -126.488, 48.605, 139.12]
  MoveL 549 to (315.56, 65.65, -151.21) mm, rotated rx -179.9 ry 0 rz -90 deg; joints [37.018, -67.033, 102.224, -126.587, 48.56, 139.195]
  MoveL 550 to (314.04, 65.58, -152.78) mm, rotated rx -179.9 ry 0 rz -90 deg; joints [36.932, -67.009, 102.198, -126.672, 48.502, 139.249]
  MoveL 551 to (313.18, 65.5, -154.79) mm, rotated rx -179.9 ry 0 rz -90 deg; joints [36.856, -66.94, 102.106, -126.733, 48.44, 139.274]
  MoveL 552 to (313.1, 65.42, -156.97) mm, rotated rx -179.9 ry 0 rz -90 deg; joints [36.801, -66.833, 101.961, -126.761, 48.38, 139.269]
  MoveL 553 to (313.79, 65.35, -159.04) mm, rotated rx -179.9 ry 0 rz -90 deg; joints [36.774, -66.703, 101.782, -126.753, 48.333, 139.234]
  MoveL 554 to (315.18, 65.27, -160.73) mm, rotated rx -179.9 ry 0 rz -90 deg; joints [36.778, -66.567, 101.593, -126.711, 48.304, 139.174]
  MoveL 555 to (317.08, 65.19, -161.81) mm, rotated rx -179.9 ry 0 rz -90 deg; joints [36.812, -66.442, 101.418, -126.641, 48.297, 139.098]
  MoveL 556 to (319.24, 65.12, -162.15) mm, rotated rx -179.9 ry 0 rz -90 deg; joints [36.873, -66.344, 101.282, -126.552, 48.314, 139.017]
  MoveL 557 to (321.38, 65.04, -161.69) mm, rotated rx -179.9 ry 0 rz -90 deg; joints [36.951, -66.286, 101.202, -126.458, 48.353, 138.943]
  MoveL 558 to (323.21, 64.96, -160.5) mm, rotated rx -179.9 ry 0 rz -90 deg; joints [37.038, -66.275, 101.19, -126.37, 48.409, 138.885]
  MoveL 559 to (324.5, 64.88, -158.74) mm, rotated rx -179.9 ry 0 rz -90 deg; joints [37.121, -66.312, 101.247, -126.301, 48.476, 138.853]
  MoveL 560 to (325.08, 64.81, -156.63) mm, rotated rx -179.9 ry 0 rz -90 deg; joints [37.189, -66.392, 101.366, -126.26, 48.544, 138.851]
  MoveL 561 to (324.87, 64.73, -154.46) mm, rotated rx -179.9 ry 0 rz -90 deg; joints [37.235, -66.505, 101.533, -126.253, 48.606, 138.879]
  MoveL 562 to (323.9, 64.65, -152.5) mm, rotated rx -179.9 ry 0 rz -90 deg; joints [37.252, -66.635, 101.724, -126.28, 48.654, 138.935]
  MoveL 563 to (322.29, 64.58, -151.02) mm, rotated rx -179.9 ry 0 rz -90 deg; joints [37.237, -66.764, 101.916, -126.339, 48.681, 139.011]
  MoveL 564 to (320.26, 64.5, -150.2) mm, rotated rx -179.9 ry 0 rz -90 deg; joints [37.192, -66.877, 102.084, -126.423, 48.684, 139.1]
  MoveL 565 to (318.08, 64.42, -150.17) mm, rotated rx -179.9 ry 0 rz -90 deg; joints [37.124, -66.957, 102.206, -126.521, 48.664, 139.189]
  MoveL 566 to (316.02, 64.35, -150.91) mm, rotated rx -179.9 ry 0 rz -90 deg; joints [37.04, -66.994, 102.267, -126.622, 48.624, 139.268]
  MoveL 567 to (314.37, 64.27, -152.33) mm, rotated rx -179.9 ry 0 rz -90 deg; joints [36.953, -66.983, 102.258, -126.712, 48.568, 139.328]
  MoveL 568 to (313.33, 64.19, -154.26) mm, rotated rx -179.9 ry 0 rz -90 deg; joints [36.874, -66.924, 102.182, -126.779, 48.506, 139.361]
  MoveL 569 to (313.04, 64.12, -156.42) mm, rotated rx -179.9 ry 0 rz -90 deg; joints [36.813, -66.826, 102.049, -126.816, 48.445, 139.363]
  MoveL 570 to (313.55, 64.04, -158.55) mm, rotated rx -179.9 ry 0 rz -90 deg; joints [36.779, -66.7, 101.876, -126.817, 48.394, 139.335]
  MoveL 571 to (314.78, 63.96, -160.36) mm, rotated rx -179.9 ry 0 rz -90 deg; joints [36.775, -66.564, 101.687, -126.784, 48.36, 139.281]
  MoveL 572 to (316.57, 63.89, -161.61) mm, rotated rx -179.9 ry 0 rz -90 deg; joints [36.802, -66.435, 101.506, -126.72, 48.347, 139.208]
  MoveL 573 to (318.69, 63.81, -162.14) mm, rotated rx -179.9 ry 0 rz -90 deg; joints [36.856, -66.329, 101.359, -126.635, 48.358, 139.127]
  MoveL 574 to (320.86, 63.73, -161.88) mm, rotated rx -179.9 ry 0 rz -90 deg; joints [36.931, -66.26, 101.263, -126.541, 48.391, 139.05]
  MoveL 575 to (322.79, 63.66, -160.86) mm, rotated rx -179.9 ry 0 rz -90 deg; joints [37.016, -66.237, 101.234, -126.45, 48.444, 138.988]
  MoveL 576 to (324.24, 63.58, -159.23) mm, rotated rx -179.9 ry 0 rz -90 deg; joints [37.101, -66.262, 101.273, -126.375, 48.508, 138.948]
  MoveL 577 to (325.01, 63.5, -157.18) mm, rotated rx -179.9 ry 0 rz -90 deg; joints [37.175, -66.332, 101.378, -126.327, 48.577, 138.938]
  MoveL 578 to (325, 63.43, -155) mm, rotated rx -179.9 ry 0 rz -90 deg; joints [37.227, -66.437, 101.534, -126.31, 48.642, 138.959]
  MoveL 579 to (324.21, 63.35, -152.96) mm, rotated rx -179.9 ry 0 rz -90 deg; joints [37.251, -66.564, 101.722, -126.329, 48.694, 139.008]
  MoveL 580 to (322.75, 63.27, -151.34) mm, rotated rx -179.9 ry 0 rz -90 deg; joints [37.244, -66.696, 101.916, -126.381, 48.726, 139.08]
  MoveL 581 to (320.8, 63.2, -150.34) mm, rotated rx -179.9 ry 0 rz -90 deg; joints [37.206, -66.814, 102.092, -126.459, 48.736, 139.166]
  MoveL 582 to (318.63, 63.12, -150.1) mm, rotated rx -179.9 ry 0 rz -90 deg; joints [37.143, -66.903, 102.228, -126.555, 48.722, 139.256]
  MoveL 583 to (316.51, 63.04, -150.65) mm, rotated rx -179.9 ry 0 rz -90 deg; joints [37.063, -66.952, 102.305, -126.656, 48.686, 139.339]
  MoveL 584 to (314.74, 62.97, -151.92) mm, rotated rx -179.9 ry 0 rz -90 deg; joints [36.976, -66.953, 102.314, -126.749, 48.634, 139.404]
  MoveL 585 to (313.52, 62.89, -153.74) mm, rotated rx -179.9 ry 0 rz -90 deg; joints [36.894, -66.906, 102.254, -126.824, 48.573, 139.445]
  MoveL 586 to (313.04, 62.81, -155.87) mm, rotated rx -179.9 ry 0 rz -90 deg; joints [36.827, -66.816, 102.134, -126.869, 48.511, 139.455]
  MoveL 587 to (313.35, 62.74, -158.03) mm, rotated rx -179.9 ry 0 rz -90 deg; joints [36.785, -66.696, 101.969, -126.879, 48.457, 139.434]
  MoveL 588 to (314.4, 62.66, -159.94) mm, rotated rx -179.9 ry 0 rz -90 deg; joints [36.773, -66.561, 101.782, -126.854, 48.417, 139.386]
  MoveL 589 to (316.07, 62.58, -161.35) mm, rotated rx -179.9 ry 0 rz -90 deg; joints [36.793, -66.429, 101.597, -126.797, 48.399, 139.317]
  MoveL 590 to (318.14, 62.51, -162.08) mm, rotated rx -179.9 ry 0 rz -90 deg; joints [36.841, -66.316, 101.438, -126.717, 48.403, 139.237]
  MoveL 591 to (320.32, 62.43, -162.02) mm, rotated rx -179.9 ry 0 rz -90 deg; joints [36.911, -66.237, 101.328, -126.624, 48.431, 139.158]
  MoveL 592 to (322.34, 62.35, -161.19) mm, rotated rx -179.9 ry 0 rz -90 deg; joints [36.995, -66.201, 101.281, -126.531, 48.479, 139.091]
  MoveL 593 to (323.93, 62.28, -159.69) mm, rotated rx -179.9 ry 0 rz -90 deg; joints [37.081, -66.214, 101.304, -126.451, 48.541, 139.045]
  MoveL 594 to (324.88, 62.2, -157.72) mm, rotated rx -179.9 ry 0 rz -90 deg; joints [37.158, -66.274, 101.393, -126.395, 48.61, 139.027]
  MoveL 595 to (325.07, 62.12, -155.55) mm, rotated rx -179.9 ry 0 rz -90 deg; joints [37.217, -66.371, 101.538, -126.37, 48.676, 139.04]
  MoveL 596 to (324.48, 62.05, -153.44) mm, rotated rx -179.9 ry 0 rz -90 deg; joints [37.248, -66.494, 101.72, -126.38, 48.732, 139.083]
  MoveL 597 to (323.17, 61.97, -151.69) mm, rotated rx -179.9 ry 0 rz -90 deg; joints [37.249, -66.626, 101.915, -126.423, 48.77, 139.15]
  MoveL 598 to (321.32, 61.89, -150.52) mm, rotated rx -179.9 ry 0 rz -90 deg; joints [37.219, -66.749, 102.098, -126.496, 48.786, 139.234]
  MoveL 599 to (319.18, 61.82, -150.09) mm, rotated rx -179.9 ry 0 rz -90 deg; joints [37.162, -66.847, 102.245, -126.588, 48.778, 139.323]
  MoveL 600 to (317.03, 61.74, -150.44) mm, rotated rx -179.9 ry 0 rz -90 deg; joints [37.085, -66.907, 102.338, -126.689, 48.748, 139.409]
  MoveL 601 to (315.14, 61.66, -151.54) mm, rotated rx -179.9 ry 0 rz -90 deg; joints [36.998, -66.92, 102.365, -126.786, 48.699, 139.479]
  MoveL 602 to (313.77, 61.59, -153.24) mm, rotated rx -179.9 ry 0 rz -90 deg; joints [36.914, -66.884, 102.322, -126.866, 48.64, 139.527]
  MoveL 603 to (313.09, 61.51, -155.32) mm, rotated rx -179.9 ry 0 rz -90 deg; joints [36.842, -66.805, 102.216, -126.919, 48.577, 139.545]
  MoveL 604 to (313.2, 61.43, -157.5) mm, rotated rx -179.9 ry 0 rz -90 deg; joints [36.794, -66.691, 102.061, -126.939, 48.52, 139.532]
  MoveL 605 to (314.07, 61.36, -159.5) mm, rotated rx -179.9 ry 0 rz -90 deg; joints [36.774, -66.559, 101.877, -126.923, 48.476, 139.49]
  MoveL 606 to (315.61, 61.28, -161.06) mm, rotated rx -179.9 ry 0 rz -90 deg; joints [36.786, -66.424, 101.688, -126.873, 48.452, 139.425]
  MoveL 607 to (317.59, 61.2, -161.97) mm, rotated rx -179.9 ry 0 rz -90 deg; joints [36.827, -66.305, 101.521, -126.798, 48.45, 139.347]
  MoveL 608 to (319.77, 61.13, -162.11) mm, rotated rx -179.9 ry 0 rz -90 deg; joints [36.893, -66.216, 101.397, -126.706, 48.473, 139.267]
  MoveL 609 to (321.86, 61.05, -161.46) mm, rotated rx -179.9 ry 0 rz -90 deg; joints [36.974, -66.169, 101.334, -126.612, 48.516, 139.196]
  MoveL 610 to (323.58, 60.97, -160.12) mm, rotated rx -179.9 ry 0 rz -90 deg; joints [37.061, -66.169, 101.338, -126.528, 48.575, 139.144]
  MoveL 611 to (324.71, 60.9, -158.25) mm, rotated rx -179.9 ry 0 rz -90 deg; joints [37.141, -66.218, 101.412, -126.465, 48.643, 139.118]
  MoveL 612 to (325.1, 60.82, -156.1) mm, rotated rx -179.9 ry 0 rz -90 deg; joints [37.205, -66.306, 101.544, -126.432, 48.711, 139.124]
  MoveL 613 to (324.7, 60.74, -153.95) mm, rotated rx -179.9 ry 0 rz -90 deg; joints [37.244, -66.424, 101.718, -126.433, 48.77, 139.159]
  MoveL 614 to (323.56, 60.67, -152.09) mm, rotated rx -179.9 ry 0 rz -90 deg; joints [37.253, -66.555, 101.912, -126.468, 48.813, 139.221]
  MoveL 615 to (321.83, 60.59, -150.75) mm, rotated rx -179.9 ry 0 rz -90 deg; joints [37.23, -66.682, 102.101, -126.534, 48.835, 139.301]
  MoveL 616 to (319.74, 60.51, -150.12) mm, rotated rx -179.9 ry 0 rz -90 deg; joints [37.179, -66.788, 102.259, -126.622, 48.833, 139.39]
  MoveL 617 to (317.56, 60.44, -150.28) mm, rotated rx -179.9 ry 0 rz -90 deg; joints [37.106, -66.858, 102.368, -126.722, 48.808, 139.478]
  MoveL 618 to (315.58, 60.36, -151.2) mm, rotated rx -179.9 ry 0 rz -90 deg; joints [37.021, -66.884, 102.412, -126.821, 48.764, 139.553]
  MoveL 619 to (314.05, 60.28, -152.77) mm, rotated rx -179.9 ry 0 rz -90 deg; joints [36.935, -66.86, 102.386, -126.907, 48.706, 139.606]
  MoveL 620 to (313.19, 60.21, -154.77) mm, rotated rx -179.9 ry 0 rz -90 deg; joints [36.859, -66.791, 102.295, -126.968, 48.644, 139.632]
  MoveL 621 to (313.09, 60.13, -156.96) mm, rotated rx -179.9 ry 0 rz -90 deg; joints [36.804, -66.685, 102.15, -126.996, 48.585, 139.627]
  MoveL 622 to (313.78, 60.05, -159.03) mm, rotated rx -179.9 ry 0 rz -90 deg; joints [36.777, -66.556, 101.971, -126.989, 48.537, 139.592]
  MoveL 623 to (315.17, 59.97, -160.72) mm, rotated rx -179.9 ry 0 rz -90 deg; joints [36.78, -66.42, 101.782, -126.947, 48.507, 139.532]
  MoveL 624 to (317.06, 59.9, -161.81) mm, rotated rx -179.9 ry 0 rz -90 deg; joints [36.815, -66.295, 101.607, -126.877, 48.499, 139.457]
  MoveL 625 to (319.22, 59.82, -162.15) mm, rotated rx -179.9 ry 0 rz -90 deg; joints [36.875, -66.197, 101.47, -126.789, 48.515, 139.376]
  MoveL 626 to (321.36, 59.74, -161.7) mm, rotated rx -179.9 ry 0 rz -90 deg; joints [36.953, -66.139, 101.39, -126.694, 48.554, 139.301]
  MoveL 627 to (323.2, 59.67, -160.52) mm, rotated rx -179.9 ry 0 rz -90 deg; joints [37.04, -66.128, 101.377, -126.606, 48.609, 139.244]
  MoveL 628 to (324.49, 59.59, -158.76) mm, rotated rx -179.9 ry 0 rz -90 deg; joints [37.123, -66.164, 101.434, -126.537, 48.676, 139.211]
  MoveL 629 to (325.08, 59.51, -156.65) mm, rotated rx -179.9 ry 0 rz -90 deg; joints [37.192, -66.244, 101.552, -126.495, 48.744, 139.209]
  MoveL 630 to (324.87, 59.44, -154.48) mm, rotated rx -179.9 ry 0 rz -90 deg; joints [37.237, -66.355, 101.718, -126.487, 48.806, 139.237]
  MoveL 631 to (323.91, 59.36, -152.52) mm, rotated rx -179.9 ry 0 rz -90 deg; joints [37.254, -66.485, 101.91, -126.514, 48.854, 139.292]
  MoveL 632 to (322.31, 59.28, -151.03) mm, rotated rx -179.9 ry 0 rz -90 deg; joints [37.24, -66.614, 102.102, -126.573, 48.882, 139.369]
  MoveL 633 to (320.28, 59.21, -150.21) mm, rotated rx -179.9 ry 0 rz -90 deg; joints [37.195, -66.727, 102.27, -126.657, 48.886, 139.456]
  MoveL 634 to (318.1, 59.13, -150.16) mm, rotated rx -179.9 ry 0 rz -90 deg; joints [37.127, -66.807, 102.392, -126.755, 48.867, 139.545]
  MoveL 635 to (316.04, 59.05, -150.9) mm, rotated rx -179.9 ry 0 rz -90 deg; joints [37.044, -66.844, 102.454, -126.855, 48.827, 139.625]
  MoveL 636 to (314.38, 58.98, -152.32) mm, rotated rx -179.9 ry 0 rz -90 deg; joints [36.957, -66.833, 102.446, -126.945, 48.773, 139.684]
  MoveL 637 to (313.34, 58.9, -154.24) mm, rotated rx -179.9 ry 0 rz -90 deg; joints [36.878, -66.775, 102.37, -127.013, 48.711, 139.718]
  MoveL 638 to (313.04, 58.82, -156.4) mm, rotated rx -179.9 ry 0 rz -90 deg; joints [36.816, -66.677, 102.237, -127.051, 48.65, 139.72]
  MoveL 639 to (313.54, 58.75, -158.53) mm, rotated rx -179.9 ry 0 rz -90 deg; joints [36.781, -66.552, 102.065, -127.053, 48.598, 139.692]
  MoveL 640 to (314.76, 58.67, -160.34) mm, rotated rx -179.9 ry 0 rz -90 deg; joints [36.777, -66.416, 101.875, -127.019, 48.563, 139.638]
  MoveL 641 to (316.55, 58.59, -161.6) mm, rotated rx -179.9 ry 0 rz -90 deg; joints [36.804, -66.287, 101.695, -126.956, 48.55, 139.566]
  MoveL 642 to (318.67, 58.52, -162.14) mm, rotated rx -179.9 ry 0 rz -90 deg; joints [36.858, -66.181, 101.546, -126.871, 48.56, 139.485]
  MoveL 643 to (320.84, 58.44, -161.88) mm, rotated rx -179.9 ry 0 rz -90 deg; joints [36.933, -66.112, 101.451, -126.776, 48.593, 139.408]
  MoveL 644 to (322.78, 58.36, -160.88) mm, rotated rx -179.9 ry 0 rz -90 deg; joints [37.018, -66.089, 101.42, -126.686, 48.644, 139.345]
  MoveL 645 to (324.23, 58.29, -159.24) mm, rotated rx -179.9 ry 0 rz -90 deg; joints [37.103, -66.113, 101.459, -126.611, 48.709, 139.306]
  MoveL 646 to (325, 58.21, -157.2) mm, rotated rx -179.9 ry 0 rz -90 deg; joints [37.177, -66.183, 101.564, -126.561, 48.777, 139.295]
  MoveL 647 to (325, 58.13, -155.02) mm, rotated rx -179.9 ry 0 rz -90 deg; joints [37.229, -66.288, 101.719, -126.544, 48.842, 139.316]
  MoveL 648 to (324.22, 58.06, -152.98) mm, rotated rx -179.9 ry 0 rz -90 deg; joints [37.254, -66.414, 101.907, -126.562, 48.894, 139.365]
  MoveL 649 to (322.76, 57.98, -151.35) mm, rotated rx -179.9 ry 0 rz -90 deg; joints [37.247, -66.545, 102.101, -126.614, 48.928, 139.437]
  MoveL 650 to (320.82, 57.9, -150.34) mm, rotated rx -179.9 ry 0 rz -90 deg; joints [37.21, -66.663, 102.278, -126.692, 48.938, 139.523]
  MoveL 651 to (318.65, 57.83, -150.1) mm, rotated rx -179.9 ry 0 rz -90 deg; joints [37.147, -66.753, 102.413, -126.787, 48.925, 139.613]
  MoveL 652 to (316.53, 57.75, -150.64) mm, rotated rx -179.9 ry 0 rz -90 deg; joints [37.066, -66.801, 102.491, -126.889, 48.89, 139.695]
  MoveL 653 to (314.75, 57.67, -151.91) mm, rotated rx -179.9 ry 0 rz -90 deg; joints [36.979, -66.803, 102.501, -126.982, 48.839, 139.761]
  MoveL 654 to (313.53, 57.6, -153.72) mm, rotated rx -179.9 ry 0 rz -90 deg; joints [36.897, -66.756, 102.442, -127.057, 48.778, 139.801]
  MoveL 655 to (313.04, 57.52, -155.85) mm, rotated rx -179.9 ry 0 rz -90 deg; joints [36.83, -66.667, 102.322, -127.103, 48.716, 139.811]
  MoveL 656 to (313.34, 57.44, -158.01) mm, rotated rx -179.9 ry 0 rz -90 deg; joints [36.788, -66.548, 102.157, -127.114, 48.661, 139.791]
  MoveL 657 to (314.39, 57.37, -159.93) mm, rotated rx -179.9 ry 0 rz -90 deg; joints [36.776, -66.413, 101.97, -127.089, 48.621, 139.743]
  MoveL 658 to (316.06, 57.29, -161.34) mm, rotated rx -179.9 ry 0 rz -90 deg; joints [36.795, -66.281, 101.784, -127.032, 48.602, 139.674]
  MoveL 659 to (318.12, 57.21, -162.07) mm, rotated rx -179.9 ry 0 rz -90 deg; joints [36.843, -66.168, 101.626, -126.952, 48.606, 139.594]
  MoveL 660 to (320.3, 57.14, -162.02) mm, rotated rx -179.9 ry 0 rz -90 deg; joints [36.913, -66.088, 101.515, -126.859, 48.633, 139.515]
  MoveL 661 to (322.32, 57.06, -161.2) mm, rotated rx -179.9 ry 0 rz -90 deg; joints [36.997, -66.053, 101.468, -126.766, 48.68, 139.448]
  MoveL 662 to (323.92, 56.98, -159.7) mm, rotated rx -179.9 ry 0 rz -90 deg; joints [37.083, -66.065, 101.489, -126.686, 48.742, 139.402]
  MoveL 663 to (324.88, 56.91, -157.74) mm, rotated rx -179.9 ry 0 rz -90 deg; joints [37.16, -66.124, 101.578, -126.629, 48.811, 139.384]
  MoveL 664 to (325.08, 56.83, -155.56) mm, rotated rx -179.9 ry 0 rz -90 deg; joints [37.219, -66.221, 101.723, -126.603, 48.877, 139.397]
  MoveL 665 to (324.48, 56.75, -153.46) mm, rotated rx -179.9 ry 0 rz -90 deg; joints [37.251, -66.343, 101.904, -126.613, 48.933, 139.439]
  MoveL 666 to (323.18, 56.68, -151.71) mm, rotated rx -179.9 ry 0 rz -90 deg; joints [37.252, -66.475, 102.099, -126.656, 48.972, 139.506]
  MoveL 667 to (321.34, 56.6, -150.53) mm, rotated rx -179.9 ry 0 rz -90 deg; joints [37.222, -66.598, 102.282, -126.728, 48.988, 139.589]
  MoveL 668 to (319.2, 56.52, -150.09) mm, rotated rx -179.9 ry 0 rz -90 deg; joints [37.165, -66.696, 102.43, -126.82, 48.981, 139.679]
  MoveL 669 to (317.04, 56.45, -150.43) mm, rotated rx -179.9 ry 0 rz -90 deg; joints [37.088, -66.756, 102.524, -126.921, 48.952, 139.764]
  MoveL 670 to (315.15, 56.37, -151.53) mm, rotated rx -179.9 ry 0 rz -90 deg; joints [37.002, -66.769, 102.551, -127.018, 48.904, 139.835]
  MoveL 671 to (313.78, 56.29, -153.22) mm, rotated rx -179.9 ry 0 rz -90 deg; joints [36.917, -66.734, 102.509, -127.099, 48.845, 139.882]
  MoveL 672 to (313.09, 56.22, -155.3) mm, rotated rx -179.9 ry 0 rz -90 deg; joints [36.846, -66.655, 102.403, -127.152, 48.782, 139.9]
  MoveL 673 to (313.19, 56.14, -157.48) mm, rotated rx -179.9 ry 0 rz -90 deg; joints [36.797, -66.542, 102.248, -127.173, 48.725, 139.888]
  MoveL 674 to (314.06, 56.06, -159.48) mm, rotated rx -179.9 ry 0 rz -90 deg; joints [36.777, -66.41, 102.064, -127.157, 48.681, 139.846]
  MoveL 675 to (315.59, 55.99, -161.05) mm, rotated rx -179.9 ry 0 rz -90 deg; joints [36.788, -66.275, 101.876, -127.108, 48.656, 139.781]
  MoveL 676 to (317.57, 55.91, -161.96) mm, rotated rx -179.9 ry 0 rz -90 deg; joints [36.829, -66.156, 101.708, -127.032, 48.653, 139.703]
  MoveL 677 to (319.75, 55.83, -162.11) mm, rotated rx -179.9 ry 0 rz -90 deg; joints [36.895, -66.067, 101.584, -126.941, 48.675, 139.623]
  MoveL 678 to (321.84, 55.76, -161.47) mm, rotated rx -179.9 ry 0 rz -90 deg; joints [36.976, -66.02, 101.519, -126.847, 48.717, 139.552]
  MoveL 679 to (323.57, 55.68, -160.13) mm, rotated rx -179.9 ry 0 rz -90 deg; joints [37.063, -66.02, 101.524, -126.762, 48.776, 139.5]
  MoveL 680 to (324.7, 55.6, -158.27) mm, rotated rx -179.9 ry 0 rz -90 deg; joints [37.143, -66.068, 101.596, -126.699, 48.843, 139.474]
  MoveL 681 to (325.1, 55.52, -156.12) mm, rotated rx -179.9 ry 0 rz -90 deg; joints [37.207, -66.156, 101.728, -126.665, 48.911, 139.479]
  MoveL 682 to (325.1, 55.53, -1) mm, rotated rx -179.9 ry 0 rz -90 deg; joints [41.275, -73.504, 111.78, -124.468, 53.128, 139.874]
  MoveL 683 to (-325.1, 55.52, -1) mm, rotated rx -179.9 ry 0 rz -90 deg; joints [12.681, -92.924, 134.073, -160.786, 41.82, 165.863]
  MoveL 684 to (-325.1, 55.52, -311.23) mm, rotated rx -179.9 ry 0 rz -90 deg; joints [9.711, -73.326, 112.126, -164.425, 38.897, 168.132]
  MoveL 685 to (325.1, 55.52, -311.23) mm, rotated rx -179.9 ry 0 rz -90 deg; joints [33.778, -58.266, 89.932, -127.237, 44.281, 137.549]
  MoveL 686 to (325.1, 55.52, -156.12) mm, rotated rx -179.9 ry 0 rz -90 deg; joints [37.207, -66.156, 101.728, -126.665, 48.911, 139.479]
  MoveC 687 to (323.81, 55.52, -151.87) mm, rotated rx -179.9 ry 0 rz -90 deg; joints [37.269, -66.411, 102.094, -126.68, 49.018, 139.558] to (320.39, 55.52, -149.05) mm, rotated rx -179.9 ry 0 rz -90 deg; joints [37.228, -66.674, 102.474, -126.802, 49.061, 139.707]
  MoveL 688 to (320.39, 55.52, -149.05) mm, rotated rx -179.9 ry 0 rz -90 deg; joints [37.228, -66.674, 102.474, -126.802, 49.061, 139.707]
  MoveC 689 to (316.96, 55.53, -146.23) mm, rotated rx -179.9 ry 0 rz -90 deg; joints [37.188, -66.938, 102.852, -126.922, 49.104, 139.855] to (315.68, 55.53, -141.98) mm, rotated rx -179.9 ry 0 rz -90 deg; joints [37.25, -67.192, 103.214, -126.934, 49.209, 139.929]
  MoveL 690 to (315.68, 55.53, -141.98) mm, rotated rx -179.9 ry 0 rz -90 deg; joints [37.25, -67.192, 103.214, -126.934, 49.209, 139.929]
  MoveL 691 to (315.68, 55.53, -14.28) mm, rotated rx -179.9 ry 0 rz -90 deg; joints [40.592, -73.264, 111.48, -125.085, 52.653, 140.196]
  MoveC 692 to (314.55, 55.53, -11.55) mm, rotated rx -179.9 ry 0 rz -90 deg; joints [40.631, -73.435, 111.705, -125.08, 52.71, 140.228] to (311.82, 55.53, -10.43) mm, rotated rx -179.9 ry 0 rz -90 deg; joints [40.574, -73.595, 111.917, -125.168, 52.703, 140.314]
  MoveL 693 to (311.82, 55.53, -10.43) mm, rotated rx -179.9 ry 0 rz -90 deg; joints [40.574, -73.595, 111.917, -125.168, 52.703, 140.314]
  MoveL 694 to (-311.82, 55.53, -10.43) mm, rotated rx -179.9 ry 0 rz -90 deg; joints [13.284, -92.076, 133.277, -159.932, 42.022, 165.249]
  MoveC 695 to (-314.55, 55.52, -11.55) mm, rotated rx -179.9 ry 0 rz -90 deg; joints [13.123, -92.042, 133.247, -160.167, 41.984, 165.422] to (-315.68, 55.52, -14.28) mm, rotated rx -179.9 ry 0 rz -90 deg; joints [13.027, -91.875, 133.091, -160.309, 41.97, 165.528]
